COMM SREFP 3 C00296 BC00296  +REFP EC00296
COMM CALL JOB:SEARCH-R1-S13D
COMM SET P032 P006
COMM SFTON3D P032
COMM SMOVL C00297 BC00297 V=166.7  +MOVJ EC00297
COMM SREFP 3 C00298 BC00298  +REFP EC00298
COMM CALL JOB:SEARCH-R1-S13D
COMM SET P032 P006
COMM SFTON3D P032
COMM SMOVL C00299 BC00299 V=166.7  +MOVJ EC00299
COMM SMOVL C00300 BC00300 V=250.0  +MOVJ EC00300
COMM SMOVL C00301 BC00301 V=166.7  +MOVJ EC00301
COMM SREFP 3 C00302 BC00302  +REFP EC00302
COMM CALL JOB:SEARCH-R1-S13D
COMM SET P032 P006
COMM SFTON3D P032
COMM SMOVL C00303 BC00303 V=166.7  +MOVJ EC00303
COMM MOVL C00304 BC00304 V=1000.0  +MOVJ EC00304 VJ=100.00
COMM 'EndPath S4107
COMM '
COMM MOVJ C00305 BC00305 VJ=100.00  +MOVJ EC00305 VJ=100.00
COMM 'Path S4208
COMM SFTOF3D
COMM MOVJ C00306 BC00306 VJ=100.00  +MOVJ EC00306 VJ=100.00
COMM MOVL C00307 BC00307 V=666.7  +MOVJ EC00307 VJ=100.00
COMM SMOVL C00308 BC00308 V=166.7  +MOVJ EC00308
COMM SREFP 3 C00309 BC00309  +REFP EC00309
COMM CALL JOB:SEARCH-R1-S13D
COMM SET P052 P006
COMM SFTON3D P052
COMM SMOVL C00310 BC00310 V=166.7  +MOVJ EC00310
COMM SREFP 3 C00311 BC00311  +REFP EC00311
COMM CALL JOB:SEARCH-R1-S13D
COMM SET P052 P006
COMM SFTON3D P052
COMM SMOVL C00312 BC00312 V=166.7  +MOVJ EC00312
COMM SFTOF3D
COMM MOVL C00313 BC00313 V=1000.0  +MOVJ EC00313 VJ=100.00
COMM SMOVL C00314 BC00314 V=500.0  +MOVJ EC00314
COMM SMOVL C00315 BC00315 V=166.7  +MOVJ EC00315
COMM SREFP 3 C00316 BC00316  +REFP EC00316
COMM CALL JOB:SEARCH-R1-S13D
COMM SET P088 P006
COMM SFTON3D P088
COMM SMOVL C00317 BC00317 V=166.7  +MOVJ EC00317
COMM SMOVL C00318 BC00318 V=166.7  +MOVJ EC00318
COMM SMOVL C00319 BC00319 V=166.7  +MOVJ EC00319
COMM SREFP 3 C00320 BC00320  +REFP EC00320
COMM CALL JOB:SEARCH-R1-S13D
COMM SET P088 P006
COMM SFTON3D P088
COMM SMOVL C00321 BC00321 V=333.3  +MOVJ EC00321
COMM SMOVL C00322 BC00322 V=666.7  +MOVJ EC00322
COMM SFTOF3D
COMM 'EndPath S4208
COMM MOVJ C00323 BC00323 VJ=100.00  +MOVJ EC00323 VJ=100.00
COMM 'Path S4209
COMM SFTOF3D
COMM MOVJ C00324 BC00324 VJ=100.00  +MOVJ EC00324 VJ=100.00
COMM MOVL C00325 BC00325 V=666.7  +MOVJ EC00325 VJ=100.00
COMM SMOVL C00326 BC00326 V=166.7  +MOVJ EC00326
COMM SREFP 3 C00327 BC00327  +REFP EC00327
COMM CALL JOB:SEARCH-R1-S13D
COMM SET P053 P006
COMM SFTON3D P053
COMM SMOVL C00328 BC00328 V=166.7  +MOVJ EC00328
COMM SMOVL C00329 BC00329 V=166.7  +MOVJ EC00329
COMM SREFP 3 C00330 BC00330  +REFP EC00330
COMM CALL JOB:SEARCH-R1-S13D
COMM SET P053 P006
COMM SFTON3D P053
COMM SMOVL C00331 BC00331 V=166.7  +MOVJ EC00331
COMM MOVL C00332 BC00332 V=1000.0  +MOVJ EC00332 VJ=100.00
COMM 'EndPath S4209
COMM *BP1
COMM MOVJ C00333 BC00333 VJ=100.00  +MOVJ EC00333 VJ=100.00
COMM 'Path W4108
COMM SFTOF3D
COMM SFTON3D P033
COMM MOVJ C00334 BC00334 VJ=100.00  +MOVJ EC00334 VJ=100.00
COMM SMOVL C00335 BC00335 V=666.7  +MOVJ EC00335
COMM SMOVL C00336 BC00336 V=166.7 PL=0  +MOVJ EC00336
COMM MACRO1 MJ#(0) ARGF14
COMM ARCON
COMM SMOVL C00337 BC00337 V=9.2  +MOVJ EC00337
COMM ARCOF
COMM SMOVL C00338 BC00338 V=800.0  +MOVJ EC00338
COMM SMOVL C00339 BC00339 V=1000.0  +MOVJ EC00339
COMM SFTOF3D
COMM 'EndPath W4108
COMM 'Path W4109
COMM SFTOF3D
COMM MOVJ C00340 BC00340 VJ=100.00  +MOVJ EC00340 VJ=100.00
COMM MOVJ C00341 BC00341 VJ=100.00  +MOVJ EC00341 VJ=100.00
COMM 'Path W4110
COMM SFTOF3D
COMM SFTON3D P033
COMM MOVJ C00342 BC00342 VJ=100.00  +MOVJ EC00342 VJ=100.00
COMM SMOVL C00343 BC00343 V=800.0  +MOVJ EC00343
COMM SMOVL C00344 BC00344 V=133.3 PL=0  +MOVJ EC00344
COMM MACRO1 MJ#(0) ARGF9
COMM ARCON
COMM SMOVL C00345 BC00345 V=11.7  +MOVJ EC00345
COMM SMOVL C00346 BC00346 V=11.7  +MOVJ EC00346
COMM SMOVL C00347 BC00347 V=11.7  +MOVJ EC00347
COMM ARCOF
COMM SMOVL C00348 BC00348 V=800.0  +MOVJ EC00348
COMM SMOVL C00349 BC00349 V=1000.0  +MOVJ EC00349
COMM SFTOF3D
COMM 'EndPath W4110
COMM MOVJ C00350 BC00350 VJ=100.00  +MOVJ EC00350 VJ=100.00
COMM '9
COMM MOVJ C00351 BC00351 VJ=100.00  +MOVJ EC00351 VJ=100.00
COMM 'Path W4111
COMM SFTOF3D
COMM SFTON3D P026
COMM MOVJ C00352 BC00352 VJ=100.00  +MOVJ EC00352 VJ=100.00
COMM SMOVL C00353 BC00353 V=666.7  +MOVJ EC00353
COMM SMOVL C00354 BC00354 V=166.7 PL=0  +MOVJ EC00354
COMM MACRO1 MJ#(0) ARGF14
COMM ARCON
COMM SMOVL C00355 BC00355 V=9.2  +MOVJ EC00355
COMM ARCOF
COMM SMOVL C00356 BC00356 V=800.0  +MOVJ EC00356
COMM SMOVL C00357 BC00357 V=1000.0  +MOVJ EC00357
COMM SFTOF3D
COMM 'EndPath W4111
COMM 'Path W4112
COMM SFTOF3D
COMM SFTON3D P026
COMM MOVJ C00358 BC00358 VJ=100.00  +MOVJ EC00358 VJ=100.00
COMM SMOVL C00359 BC00359 V=800.0  +MOVJ EC00359
COMM SMOVL C00360 BC00360 V=150.0 PL=0  +MOVJ EC00360
COMM ARCON
COMM SMOVL C00361 BC00361 V=11.7  +MOVJ EC00361
COMM SMOVL C00362 BC00362 V=11.7  +MOVJ EC00362
COMM SMOVL C00363 BC00363 V=11.7  +MOVJ EC00363
COMM ARCOF
COMM SMOVL C00364 BC00364 V=800.0  +MOVJ EC00364
COMM SMOVL C00365 BC00365 V=1000.0  +MOVJ EC00365
COMM SFTOF3D
COMM MOVJ C00366 BC00366 VJ=100.00  +MOVJ EC00366 VJ=100.00
COMM MOVJ C00367 BC00367 VJ=100.00  +MOVJ EC00367 VJ=100.00
COMM 'uwaga na podajnik
COMM 'Path W4114
COMM SFTOF3D
COMM SFTON3D P026
COMM MOVJ C00368 BC00368 VJ=100.00  +MOVJ EC00368 VJ=100.00
COMM SMOVL C00369 BC00369 V=800.0  +MOVJ EC00369
COMM SMOVL C00370 BC00370 V=150.0 PL=0  +MOVJ EC00370
COMM ARCON
COMM SMOVL C00371 BC00371 V=11.7  +MOVJ EC00371
COMM ARCOF
COMM SMOVL C00372 BC00372 V=800.0  +MOVJ EC00372
COMM SMOVL C00373 BC00373 V=1000.0  +MOVJ EC00373
COMM SFTOF3D
COMM 'EndPath W4114
COMM 'brak dostepu offset drutu 1cm
COMM 'Path W4115
COMM SFTOF3D
COMM SFTON3D P026
COMM MOVJ C00374 BC00374 VJ=100.00  +MOVJ EC00374 VJ=100.00
COMM SMOVL C00375 BC00375 V=800.0  +MOVJ EC00375
COMM SMOVL C00376 BC00376 V=150.0 PL=0  +MOVJ EC00376
COMM ARCON
COMM SMOVL C00377 BC00377 V=11.7  +MOVJ EC00377
COMM ARCOF
COMM SMOVL C00378 BC00378 V=800.0  +MOVJ EC00378
COMM SMOVL C00379 BC00379 V=1000.0  +MOVJ EC00379
COMM SFTOF3D
COMM 'EndPath W4115
COMM MOVJ C00380 BC00380 VJ=100.00  +MOVJ EC00380 VJ=100.00
COMM '10
COMM '11
COMM MOVJ C00381 BC00381 VJ=100.00  +MOVJ EC00381 VJ=100.00
COMM 'Path W4118
COMM SFTOF3D
COMM SFTON3D P025
COMM MOVJ C00382 BC00382 VJ=100.00  +MOVJ EC00382 VJ=100.00
COMM SMOVL C00383 BC00383 V=800.0  +MOVJ EC00383
COMM SMOVL C00384 BC00384 V=166.7  +MOVJ EC00384
COMM ARCON
COMM SMOVL C00385 BC00385 V=9.2  +MOVJ EC00385
COMM SMOVL C00386 BC00386 V=9.2  +MOVJ EC00386
COMM SMOVL C00387 BC00387 V=9.2  +MOVJ EC00387
COMM SMOVL C00388 BC00388 V=9.2  +MOVJ EC00388
COMM SMOVL C00389 BC00389 V=9.2  +MOVJ EC00389
COMM ARCOF
COMM SMOVL C00390 BC00390 V=800.0  +MOVJ EC00390
COMM SMOVL C00391 BC00391 V=1000.0  +MOVJ EC00391
COMM SFTOF3D
COMM 'EndPath W4118
COMM 'brak dostepu offset drutu 1cm
COMM MOVJ C00392 BC00392 VJ=100.00  +MOVJ EC00392 VJ=100.00
COMM 'Path W4117
COMM SFTOF3D
COMM SFTON3D P025
COMM MOVJ C00393 BC00393 VJ=100.00  +MOVJ EC00393 VJ=100.00
COMM SMOVL C00394 BC00394 V=800.0  +MOVJ EC00394
COMM SMOVL C00395 BC00395 V=166.7 PL=0  +MOVJ EC00395
COMM ARCON
COMM SMOVL C00396 BC00396 V=10.0  +MOVJ EC00396
COMM ARCOF
COMM SMOVL C00397 BC00397 V=800.0  +MOVJ EC00397
COMM SMOVL C00398 BC00398 V=1000.0  +MOVJ EC00398
COMM SFTOF3D
COMM 'EndPath W4117
COMM '12
COMM MOVJ C00399 BC00399 VJ=100.00  +MOVJ EC00399 VJ=100.00
COMM MOVJ C00400 BC00400 VJ=100.00  +MOVJ EC00400 VJ=100.00
COMM 'Path W4859
COMM SFTOF3D
COMM SFTON3D P073
COMM MOVJ C00401 BC00401 VJ=100.00  +MOVJ EC00401 VJ=100.00
COMM SMOVL C00402 BC00402 V=800.0  +MOVJ EC00402
COMM SMOVL C00403 BC00403 V=150.0 PL=0  +MOVJ EC00403
COMM ARCON
COMM SMOVL C00404 BC00404 V=8.3  +MOVJ EC00404
COMM SFTON3D P074
COMM SMOVL C00405 BC00405 V=9.2  +MOVJ EC00405
COMM SMOVL C00406 BC00406 V=9.2  +MOVJ EC00406
COMM ARCOF
COMM SMOVL C00407 BC00407 V=800.0  +MOVJ EC00407
COMM SMOVL C00408 BC00408 V=1000.0  +MOVJ EC00408
COMM SFTOF3D
COMM 'EndPath W4859
COMM MOVJ C00409 BC00409 VJ=100.00  +MOVJ EC00409 VJ=100.00
COMM MOVJ C00410 BC00410 VJ=100.00  +MOVJ EC00410 VJ=100.00
COMM 'Path W4119
COMM SFTOF3D
COMM SFTON3D P034
COMM MOVJ C00411 BC00411 VJ=100.00  +MOVJ EC00411 VJ=100.00
COMM SMOVL C00412 BC00412 V=800.0  +MOVJ EC00412
COMM SMOVL C00413 BC00413 V=150.0 PL=0  +MOVJ EC00413
COMM ARCON
COMM SMOVL C00414 BC00414 V=10.0  +MOVJ EC00414
COMM SMOVL C00415 BC00415 V=10.0  +MOVJ EC00415
COMM SMOVL C00416 BC00416 V=10.0  +MOVJ EC00416
COMM ARCOF
COMM SMOVL C00417 BC00417 V=800.0  +MOVJ EC00417
COMM SMOVL C00418 BC00418 V=1000.0  +MOVJ EC00418
COMM SFTOF3D
COMM 'EndPath W4119
COMM 'Path W4210
COMM SFTOF3D
COMM SFTON3D P050
COMM MOVJ C00419 BC00419 VJ=100.00  +MOVJ EC00419 VJ=100.00
COMM SMOVL C00420 BC00420 V=800.0  +MOVJ EC00420
COMM SMOVL C00421 BC00421 V=150.0 PL=0  +MOVJ EC00421
COMM ARCON
COMM SMOVL C00422 BC00422 V=11.7  +MOVJ EC00422
COMM ARCOF
COMM SMOVL C00423 BC00423 V=800.0  +MOVJ EC00423
COMM SMOVL C00424 BC00424 V=1000.0  +MOVJ EC00424
COMM SFTOF3D
COMM 'EndPath W4210
COMM 'Path W4211
COMM SFTOF3D
COMM SFTON3D P034
COMM MOVJ C00425 BC00425 VJ=100.00  +MOVJ EC00425 VJ=100.00
COMM SMOVL C00426 BC00426 V=800.0  +MOVJ EC00426
COMM SMOVL C00427 BC00427 V=166.7 PL=0  +MOVJ EC00427
COMM ARCON
COMM SWVON WEV#(66)
COMM SMOVL C00428 BC00428 V=9.2  +MOVJ EC00428
COMM SMOVL C00429 BC00429 V=9.2  +MOVJ EC00429
COMM SMOVL C00430 BC00430 V=9.2  +MOVJ EC00430
COMM ARCOF
COMM SMOVL C00431 BC00431 V=800.0  +MOVJ EC00431
COMM SMOVL C00432 BC00432 V=1000.0  +MOVJ EC00432
COMM MOVJ C00433 BC00433 VJ=30.00  +MOVJ EC00433 VJ=30.00
COMM MOVJ C00434 BC00434 VJ=30.00  +MOVJ EC00434 VJ=30.00
COMM SFTOF3D
COMM MACRO1 MJ#(0) ARGF6
COMM MOVJ C00435 BC00435 VJ=30.00  +MOVJ EC00435 VJ=30.00
COMM SFTON3D P063
COMM SMOVL C00436 BC00436 V=133.3  +MOVJ EC00436
COMM ARCON
COMM SMOVL C00437 BC00437 V=11.7  +MOVJ EC00437
COMM SMOVL C00438 BC00438 V=11.7  +MOVJ EC00438
COMM SMOVL C00439 BC00439 V=11.7  +MOVJ EC00439
COMM SFTON3D P062
COMM SMOVL C00440 BC00440 V=11.7  +MOVJ EC00440
COMM SMOVL C00441 BC00441 V=11.7  +MOVJ EC00441
COMM SFTON3D P061
COMM SMOVL C00442 BC00442 V=11.0  +MOVJ EC00442
COMM SMOVL C00443 BC00443 V=11.0  +MOVJ EC00443
COMM ARCOF
COMM SMOVL C00444 BC00444 V=250.0  +MOVJ EC00444
COMM SFTOF3D
COMM MOVJ C00445 BC00445 VJ=30.00  +MOVJ EC00445 VJ=30.00
COMM MOVJ C00446 BC00446 VJ=30.00  +MOVJ EC00446 VJ=30.00
COMM 'EndPath W4211
COMM 'Path W4210
COMM SFTOF3D
COMM SFTON3D P054
COMM MOVJ C00447 BC00447 VJ=100.00  +MOVJ EC00447 VJ=100.00
COMM SMOVL C00448 BC00448 V=800.0  +MOVJ EC00448
COMM SMOVL C00449 BC00449 V=150.0 PL=0  +MOVJ EC00449
COMM MACRO1 MJ#(0) ARGF14
COMM ARCON
COMM SWVON WEV#(67)
COMM SMOVL C00450 BC00450 V=10.0  +MOVJ EC00450
COMM SMOVL C00451 BC00451 V=10.0  +MOVJ EC00451
COMM ARCOF
COMM SWVOF
COMM SMOVL C00452 BC00452 V=800.0  +MOVJ EC00452
COMM SMOVL C00453 BC00453 V=1000.0  +MOVJ EC00453
COMM SFTOF3D
COMM 'EndPath W4210
COMM 'Path W4121
COMM SFTOF3D
COMM SFTON3D P028
COMM MOVJ C00454 BC00454 VJ=100.00  +MOVJ EC00454 VJ=100.00
COMM SMOVL C00455 BC00455 V=800.0  +MOVJ EC00455
COMM SMOVL C00456 BC00456 V=150.0 PL=0  +MOVJ EC00456
COMM ARCON
COMM SMOVL C00457 BC00457 V=9.2  +MOVJ EC00457
COMM SMOVL C00458 BC00458 V=9.2  +MOVJ EC00458
COMM SMOVL C00459 BC00459 V=9.2  +MOVJ EC00459
COMM ARCOF
COMM SMOVL C00460 BC00460 V=800.0  +MOVJ EC00460
COMM SMOVL C00461 BC00461 V=1000.0  +MOVJ EC00461
COMM SFTOF3D
COMM 'EndPath W4121
COMM 'brak dostepu offset 5mm
COMM MOVJ C00462 BC00462 VJ=100.00  +MOVJ EC00462 VJ=100.00
COMM 'Path W4122
COMM SFTOF3D
COMM SFTON3D P028
COMM MOVJ C00463 BC00463 VJ=100.00  +MOVJ EC00463 VJ=100.00
COMM SMOVL C00464 BC00464 V=800.0  +MOVJ EC00464
COMM SMOVL C00465 BC00465 V=166.7 PL=0  +MOVJ EC00465
COMM ARCON
COMM SMOVL C00466 BC00466 V=11.7  +MOVJ EC00466
COMM ARCOF
COMM SMOVL C00467 BC00467 V=800.0  +MOVJ EC00467
COMM SMOVL C00468 BC00468 V=1000.0  +MOVJ EC00468
COMM SFTOF3D
COMM 'EndPath W4122
COMM MOVJ C00469 BC00469 VJ=100.00  +MOVJ EC00469 VJ=100.00
COMM '13
COMM MOVJ C00470 BC00470 VJ=100.00  +MOVJ EC00470 VJ=100.00
COMM 'Path W4123
COMM SFTOF3D
COMM SFTON3D P030
COMM MOVJ C00471 BC00471 VJ=100.00  +MOVJ EC00471 VJ=100.00
COMM SMOVL C00472 BC00472 V=800.0  +MOVJ EC00472
COMM SMOVL C00473 BC00473 V=150.0 PL=0  +MOVJ EC00473
COMM MACRO1 MJ#(0) ARGF9
COMM ARCON
COMM SWVON WEV#(10)
COMM SFTON3D P031
COMM SMOVL C00474 BC00474 V=12.5  +MOVJ EC00474
COMM ARCOF
COMM SWVOF
COMM SMOVL C00475 BC00475 V=800.0  +MOVJ EC00475
COMM SMOVL C00476 BC00476 V=1000.0  +MOVJ EC00476
COMM SFTOF3D
COMM 'EndPath W4123
COMM '14
COMM '15-brak
COMM 'Path W4212
COMM SFTOF3D
COMM SFTON3D P052
COMM MOVJ C00477 BC00477 VJ=100.00  +MOVJ EC00477 VJ=100.00
COMM SMOVL C00478 BC00478 V=800.0  +MOVJ EC00478
COMM SMOVL C00479 BC00479 V=150.0 PL=0  +MOVJ EC00479
COMM ARCON
COMM SMOVL C00480 BC00480 V=10.8  +MOVJ EC00480
COMM SMOVL C00481 BC00481 V=10.8  +MOVJ EC00481
COMM SMOVL C00482 BC00482 V=10.8  +MOVJ EC00482
COMM ARCOF
COMM SMOVL C00483 BC00483 V=800.0  +MOVJ EC00483
COMM MACRO1 MJ#(0) ARGF6
COMM SMOVL C00484 BC00484 V=333.3  +MOVJ EC00484
COMM SFTOF3D
COMM 'DODAC SHIFT
COMM SFTON3D P088
COMM SMOVL C00485 BC00485 V=133.3  +MOVJ EC00485
COMM ARCON
COMM SMOVL C00486 BC00486 V=10.8  +MOVJ EC00486
COMM ARCOF
COMM SMOVL C00487 BC00487 V=250.0  +MOVJ EC00487
COMM SMOVL C00488 BC00488 V=1000.0  +MOVJ EC00488
COMM SFTOF3D
COMM 'EndPath W4212
COMM '16
COMM 'Path W4213
COMM SFTOF3D
COMM SFTON3D P053
COMM MOVJ C00489 BC00489 VJ=100.00  +MOVJ EC00489 VJ=100.00
COMM SMOVL C00490 BC00490 V=800.0  +MOVJ EC00490
COMM SMOVL C00491 BC00491 V=150.0 PL=0  +MOVJ EC00491
COMM MACRO1 MJ#(0) ARGF9
COMM ARCON
COMM SMOVL C00492 BC00492 V=10.8  +MOVJ EC00492
COMM SMOVL C00493 BC00493 V=10.8  +MOVJ EC00493
COMM SMOVL C00494 BC00494 V=10.8  +MOVJ EC00494
COMM ARCOF
COMM SMOVL C00495 BC00495 V=800.0  +MOVJ EC00495
COMM SMOVL C00496 BC00496 V=1000.0  +MOVJ EC00496
COMM SFTOF3D
COMM 'EndPath W4213
COMM 'Path W4124
COMM SFTOF3D
COMM SFTON3D P029
COMM MOVJ C00497 BC00497 VJ=100.00  +MOVJ EC00497 VJ=100.00
COMM SMOVL C00498 BC00498 V=800.0  +MOVJ EC00498
COMM SMOVL C00499 BC00499 V=166.7 PL=0  +MOVJ EC00499
COMM MACRO1 MJ#(0) ARGF14
COMM ARCON
COMM SMOVL C00500 BC00500 V=10.0  +MOVJ EC00500
COMM SMOVL C00501 BC00501 V=10.0  +MOVJ EC00501
COMM ARCOF
COMM SMOVL C00502 BC00502 V=800.0  +MOVJ EC00502
COMM SMOVL C00503 BC00503 V=1000.0  +MOVJ EC00503
COMM SFTOF3D
COMM 'EndPath W4124
COMM MOVJ C00504 BC00504 VJ=100.00  +MOVJ EC00504 VJ=100.00
COMM 'Path W4125
COMM SFTOF3D
COMM SFTON3D P029
COMM MOVJ C00505 BC00505 VJ=100.00  +MOVJ EC00505 VJ=100.00
COMM SMOVL C00506 BC00506 V=800.0  +MOVJ EC00506
COMM SMOVL C00507 BC00507 V=150.0 PL=0  +MOVJ EC00507
COMM ARCON
COMM SMOVL C00508 BC00508 V=11.7  +MOVJ EC00508
COMM SMOVL C00509 BC00509 V=11.7  +MOVJ EC00509
COMM SMOVL C00510 BC00510 V=11.7  +MOVJ EC00510
COMM ARCOF
COMM SMOVL C00511 BC00511 V=800.0  +MOVJ EC00511
COMM SMOVL C00512 BC00512 V=1000.0  +MOVJ EC00512
COMM SFTOF3D
COMM 'EndPath W4125
COMM MOVJ C00513 BC00513 VJ=100.00  +MOVJ EC00513 VJ=100.00
COMM 'Path W4126
COMM SFTOF3D
COMM SFTON3D P029
COMM MOVJ C00514 BC00514 VJ=100.00  +MOVJ EC00514 VJ=100.00
COMM SMOVL C00515 BC00515 V=800.0  +MOVJ EC00515
COMM SMOVL C00516 BC00516 V=166.7 PL=0  +MOVJ EC00516
COMM ARCON
COMM SMOVL C00517 BC00517 V=11.7  +MOVJ EC00517
COMM ARCON
COMM SMOVL C00518 BC00518 V=11.7  +MOVJ EC00518
COMM SMOVL C00519 BC00519 V=11.7  +MOVJ EC00519
COMM ARCOF
COMM SMOVL C00520 BC00520 V=800.0  +MOVJ EC00520
COMM SMOVL C00521 BC00521 V=1000.0  +MOVJ EC00521
COMM SFTOF3D
COMM 'EndPath W4126
COMM MOVJ C00522 BC00522 VJ=100.00  +MOVJ EC00522 VJ=100.00
COMM '17
COMM 'Path W4127
COMM SFTOF3D
COMM SFTON3D P027
COMM MOVJ C00523 BC00523 VJ=100.00  +MOVJ EC00523 VJ=100.00
COMM SMOVL C00524 BC00524 V=800.0  +MOVJ EC00524
COMM SMOVL C00525 BC00525 V=150.0 PL=0  +MOVJ EC00525
COMM ARCON
COMM SMOVL C00526 BC00526 V=10.0  +MOVJ EC00526
COMM ARCOF
COMM SMOVL C00527 BC00527 V=800.0  +MOVJ EC00527
COMM SMOVL C00528 BC00528 V=1000.0  +MOVJ EC00528
COMM SFTOF3D
COMM 'EndPath W4127
COMM 'Path W4128
COMM SFTOF3D
COMM SFTON3D P027
COMM MOVJ C00529 BC00529 VJ=100.00  +MOVJ EC00529 VJ=100.00
COMM SMOVL C00530 BC00530 V=800.0  +MOVJ EC00530
COMM SMOVL C00531 BC00531 V=150.0 PL=0  +MOVJ EC00531
COMM ARCON
COMM SMOVL C00532 BC00532 V=11.7  +MOVJ EC00532
COMM ARCOF
COMM SMOVL C00533 BC00533 V=800.0  +MOVJ EC00533
COMM SMOVL C00534 BC00534 V=1000.0  +MOVJ EC00534
COMM SFTOF3D
COMM 'EndPath W4128
COMM 'Path W4129
COMM SFTOF3D
COMM SFTON3D P027
COMM MOVJ C00535 BC00535 VJ=100.00  +MOVJ EC00535 VJ=100.00
COMM SMOVL C00536 BC00536 V=800.0  +MOVJ EC00536
COMM SMOVL C00537 BC00537 V=150.0 PL=0  +MOVJ EC00537
COMM SMOVL C00538 BC00538 V=16.7  +MOVJ EC00538
COMM ARCOF
COMM SMOVL C00539 BC00539 V=800.0  +MOVJ EC00539
COMM SMOVL C00540 BC00540 V=1000.0  +MOVJ EC00540
COMM SFTOF3D
COMM 'EndPath W4129
COMM '18
COMM MOVJ C00541 BC00541 VJ=100.00  +MOVJ EC00541 VJ=100.00
COMM 'Path W4130
COMM SFTOF3D
COMM SFTON3D P024
COMM MOVJ C00542 BC00542 VJ=100.00  +MOVJ EC00542 VJ=100.00
COMM SMOVL C00543 BC00543 V=800.0  +MOVJ EC00543
COMM SMOVL C00544 BC00544 V=150.0 PL=0  +MOVJ EC00544
COMM ARCON
COMM SMOVL C00545 BC00545 V=9.2  +MOVJ EC00545
COMM SMOVL C00546 BC00546 V=9.2  +MOVJ EC00546
COMM SMOVL C00547 BC00547 V=9.2  +MOVJ EC00547
COMM SMOVL C00548 BC00548 V=9.2  +MOVJ EC00548
COMM ARCOF
COMM SMOVL C00549 BC00549 V=800.0  +MOVJ EC00549
COMM SMOVL C00550 BC00550 V=1000.0  +MOVJ EC00550
COMM SFTOF3D
COMM 'EndPath W4130
COMM 'Path W4860
COMM SFTOF3D
COMM SFTON3D P071
COMM MOVJ C00551 BC00551 VJ=100.00  +MOVJ EC00551 VJ=100.00
COMM SMOVL C00552 BC00552 V=800.0  +MOVJ EC00552
COMM SMOVL C00553 BC00553 V=150.0 PL=0  +MOVJ EC00553
COMM MACRO1 MJ#(0) ARGF9
COMM ARCON
COMM SMOVL C00554 BC00554 V=9.2  +MOVJ EC00554
COMM SFTON3D P072
COMM ARCON
COMM SMOVL C00555 BC00555 V=9.2  +MOVJ EC00555
COMM SMOVL C00556 BC00556 V=9.2  +MOVJ EC00556
COMM ARCOF
COMM SMOVL C00557 BC00557 V=800.0  +MOVJ EC00557
COMM SMOVL C00558 BC00558 V=1000.0  +MOVJ EC00558
COMM SFTOF3D
COMM 'EndPath W4860
COMM '19
COMM MOVJ C00559 BC00559 VJ=100.00  +MOVJ EC00559 VJ=100.00
COMM 'Path W4131
COMM SFTOF3D
COMM SFTON3D P023
COMM MOVJ C00560 BC00560 VJ=100.00  +MOVJ EC00560 VJ=100.00
COMM SMOVL C00561 BC00561 V=800.0  +MOVJ EC00561
COMM SMOVL C00562 BC00562 V=166.7 PL=0  +MOVJ EC00562
COMM MACRO1 MJ#(0) ARGF9
COMM ARCON
COMM SWVON WEV#(60)
COMM SMOVL C00563 BC00563 V=7.5  +MOVJ EC00563
COMM SMOVL C00564 BC00564 V=7.5  +MOVJ EC00564
COMM SMOVL C00565 BC00565 V=7.5  +MOVJ EC00565
COMM ARCOF
COMM SWVOF
COMM SMOVL C00566 BC00566 V=800.0  +MOVJ EC00566
COMM SMOVL C00567 BC00567 V=1000.0  +MOVJ EC00567
COMM SFTOF3D
COMM 'EndPath W4131
COMM MOVJ C00568 BC00568 VJ=100.00  +MOVJ EC00568 VJ=100.00
COMM 'Path W4214
COMM SFTOF3D
COMM SFTON3D P089
COMM MOVJ C00569 BC00569 VJ=100.00  +MOVJ EC00569 VJ=100.00
COMM SMOVL C00570 BC00570 V=800.0  +MOVJ EC00570
COMM SMOVL C00571 BC00571 V=150.0 PL=0  +MOVJ EC00571
COMM MACRO1 MJ#(0) ARGF9
COMM ARCON
COMM SMOVL C00572 BC00572 V=9.2  +MOVJ EC00572
COMM SFTON3D P050
COMM SMOVL C00573 BC00573 V=9.2  +MOVJ EC00573
COMM SMOVL C00574 BC00574 V=9.2  +MOVJ EC00574
COMM ARCOF
COMM SMOVL C00575 BC00575 V=800.0  +MOVJ EC00575
COMM SMOVL C00576 BC00576 V=1000.0  +MOVJ EC00576
COMM SFTOF3D
COMM 'EndPath W4214
COMM 'Path W4215
COMM SFTOF3D
COMM SFTON3D P051
COMM MOVJ C00577 BC00577 VJ=100.00  +MOVJ EC00577 VJ=100.00
COMM SMOVL C00578 BC00578 V=800.0  +MOVJ EC00578
COMM SMOVL C00579 BC00579 V=150.0 PL=0  +MOVJ EC00579
COMM MACRO1 MJ#(0) ARGF9
COMM ARCON
COMM SWVON WEV#(60)
COMM SMOVL C00580 BC00580 V=7.5  +MOVJ EC00580
COMM SMOVL C00581 BC00581 V=7.5  +MOVJ EC00581
COMM SMOVL C00582 BC00582 V=7.5  +MOVJ EC00582
COMM ARCOF
COMM SWVOF
COMM SMOVL C00583 BC00583 V=800.0  +MOVJ EC00583
COMM SMOVL C00584 BC00584 V=1000.0  +MOVJ EC00584
COMM SFTOF3D
COMM 'EndPath W4215
COMM MOVJ C00585 BC00585 VJ=100.00  +MOVJ EC00585 VJ=100.00
COMM '20
COMM 'offset 5mm
COMM MOVJ C00586 BC00586 VJ=100.00  +MOVJ EC00586 VJ=100.00
COMM MOVJ C00587 BC00587 VJ=100.00  +MOVJ EC00587 VJ=100.00
COMM 'Path W4132
COMM SFTOF3D
COMM SFTON3D P032
COMM MOVJ C00588 BC00588 VJ=100.00  +MOVJ EC00588 VJ=100.00
COMM SMOVL C00589 BC00589 V=800.0  +MOVJ EC00589
COMM SMOVL C00590 BC00590 V=150.0 PL=0  +MOVJ EC00590
COMM ARCON
COMM SMOVL C00591 BC00591 V=10.0  +MOVJ EC00591
COMM SMOVL C00592 BC00592 V=10.0  +MOVJ EC00592
COMM ARCOF
COMM SMOVL C00593 BC00593 V=800.0  +MOVJ EC00593
COMM SMOVL C00594 BC00594 V=1000.0  +MOVJ EC00594
COMM SFTOF3D
COMM JUMP *FFF
COMM 'EndPath W4132
COMM 'Path W4133
COMM SFTOF3D
COMM SFTON3D P032
COMM MOVJ C00595 BC00595 VJ=100.00  +MOVJ EC00595 VJ=100.00
COMM SMOVL C00596 BC00596 V=800.0  +MOVJ EC00596
COMM SMOVL C00597 BC00597 V=166.7 PL=0  +MOVJ EC00597
COMM ARCON
COMM SMOVL C00598 BC00598 V=10.0  +MOVJ EC00598
COMM ARCOF
COMM SMOVL C00599 BC00599 V=800.0  +MOVJ EC00599
COMM SMOVL C00600 BC00600 V=1000.0  +MOVJ EC00600
COMM SFTOF3D
COMM 'EndPath W4133
COMM 'Path W4134
COMM SFTOF3D
COMM SFTON3D P032
COMM MOVJ C00601 BC00601 VJ=100.00  +MOVJ EC00601 VJ=100.00
COMM SMOVL C00602 BC00602 V=800.0  +MOVJ EC00602
COMM SMOVL C00603 BC00603 V=150.0 PL=0  +MOVJ EC00603
COMM ARCON
COMM SMOVL C00604 BC00604 V=10.0  +MOVJ EC00604
COMM ARCOF
COMM SMOVL C00605 BC00605 V=800.0  +MOVJ EC00605
COMM *FFF
COMM SMOVL C00606 BC00606 V=1000.0  +MOVJ EC00606
COMM SFTOF3D
COMM 'EndPath W4134
COMM 'offset 5mm
COMM MOVJ C00607 BC00607 VJ=100.00  +MOVJ EC00607 VJ=100.00
COMM 'Path W4135
COMM SFTOF3D
COMM SFTON3D P032
COMM MOVJ C00608 BC00608 VJ=100.00  +MOVJ EC00608 VJ=100.00
COMM SMOVL C00609 BC00609 V=800.0  +MOVJ EC00609
COMM SMOVL C00610 BC00610 V=166.7 PL=0  +MOVJ EC00610
COMM ARCON
COMM SMOVL C00611 BC00611 V=10.0  +MOVJ EC00611
COMM ARCOF
COMM SMOVL C00612 BC00612 V=800.0  +MOVJ EC00612
COMM SMOVL C00613 BC00613 V=1000.0  +MOVJ EC00613
COMM SFTOF3D
COMM 'EndPath W4135
COMM MOVJ C00614 BC00614 VJ=100.00  +MOVJ EC00614 VJ=100.00
COMM 'Path W4136
COMM SFTOF3D
COMM SFTON3D P032
COMM MOVJ C00615 BC00615 VJ=100.00  +MOVJ EC00615 VJ=100.00
COMM SMOVL C00616 BC00616 V=800.0  +MOVJ EC00616
COMM SMOVL C00617 BC00617 V=166.7 PL=0  +MOVJ EC00617
COMM ARCON
COMM SMOVL C00618 BC00618 V=11.7  +MOVJ EC00618
COMM SMOVL C00619 BC00619 V=11.7  +MOVJ EC00619
COMM ARCOF
COMM SMOVL C00620 BC00620 V=800.0  +MOVJ EC00620
COMM SMOVL C00621 BC00621 V=1000.0  +MOVJ EC00621
COMM SFTOF3D
COMM 'EndPath W4136
COMM MOVJ C00622 BC00622 VJ=100.00  +MOVJ EC00622 VJ=100.00
COMM MOVJ C00623 BC00623 VJ=100.00  +MOVJ EC00623 VJ=100.00
COMM 'Path W4137
COMM SFTOF3D
COMM SFTON3D P021
COMM MOVJ C00624 BC00624 VJ=100.00  +MOVJ EC00624 VJ=100.00
COMM SMOVL C00625 BC00625 V=800.0  +MOVJ EC00625
COMM SMOVL C00626 BC00626 V=150.0 PL=0  +MOVJ EC00626
COMM MACRO1 MJ#(0) ARGF9
COMM ARCON
COMM SFTON3D P022
COMM SMOVL C00627 BC00627 V=10.0  +MOVJ EC00627
COMM ARCOF
COMM SMOVL C00628 BC00628 V=800.0  +MOVJ EC00628
COMM SMOVL C00629 BC00629 V=1000.0  +MOVJ EC00629
COMM SFTOF3D
COMM 'EndPath W4137
COMM MOVJ C00630 BC00630 VJ=100.00  +MOVJ EC00630 VJ=100.00
COMM 'Path W4724
COMM SFTOF3D
COMM SFTON3D P095
COMM MOVJ C00631 BC00631 VJ=100.00  +MOVJ EC00631 VJ=100.00
COMM SMOVL C00632 BC00632 V=800.0  +MOVJ EC00632
COMM SMOVL C00633 BC00633 V=150.0 PL=0  +MOVJ EC00633
COMM ARCON
COMM SMOVL C00634 BC00634 V=10.0  +MOVJ EC00634
COMM SMOVL C00635 BC00635 V=10.0  +MOVJ EC00635
COMM SMOVL C00636 BC00636 V=10.0  +MOVJ EC00636
COMM ARCOF
COMM SMOVL C00637 BC00637 V=800.0  +MOVJ EC00637
COMM SMOVL C00638 BC00638 V=1000.0  +MOVJ EC00638
COMM SFTOF3D
COMM 'EndPath W4724
COMM 'Path W4725
COMM SFTOF3D
COMM SFTON3D P096
COMM MOVJ C00639 BC00639 VJ=100.00  +MOVJ EC00639 VJ=100.00
COMM SMOVL C00640 BC00640 V=800.0  +MOVJ EC00640
COMM SMOVL C00641 BC00641 V=150.0 PL=0  +MOVJ EC00641
COMM ARCON
COMM SMOVL C00642 BC00642 V=10.0  +MOVJ EC00642
COMM SMOVL C00643 BC00643 V=10.0  +MOVJ EC00643
COMM ARCOF
COMM SMOVL C00644 BC00644 V=800.0  +MOVJ EC00644
COMM SMOVL C00645 BC00645 V=1000.0  +MOVJ EC00645
COMM SFTOF3D
COMM 'EndPath W4725
COMM MOVJ C00646 BC00646 VJ=100.00  +MOVJ EC00646 VJ=100.00
COMM 'Path W4861
COMM SFTOF3D
COMM SFTON3D P071
COMM MOVJ C00647 BC00647 VJ=100.00  +MOVJ EC00647 VJ=100.00
COMM SMOVL C00648 BC00648 V=800.0  +MOVJ EC00648
COMM SMOVL C00649 BC00649 V=150.0 PL=0  +MOVJ EC00649
COMM MACRO1 MJ#(0) ARGF14
COMM ARCON
COMM SMOVL C00650 BC00650 V=9.2  +MOVJ EC00650
COMM SFTON3D P073
COMM SMOVL C00651 BC00651 V=9.2  +MOVJ EC00651
COMM SMOVL C00652 BC00652 V=9.2  +MOVJ EC00652
COMM ARCOF
COMM SMOVL C00653 BC00653 V=800.0  +MOVJ EC00653
COMM SMOVL C00654 BC00654 V=1000.0  +MOVJ EC00654
COMM SFTOF3D
COMM 'EndPath W4861
COMM MOVJ C00655 BC00655 VJ=100.00  +MOVJ EC00655 VJ=100.00
COMM MOVJ C00656 BC00656 VJ=100.00  +MOVJ EC00656 VJ=100.00
'X2_8B-21B(90,180)
'
MOVJ C00657 BC00657 VJ=100.00  +MOVJ EC00657 VJ=100.00
'Path S4722
SFTOF3D
MOVJ C00658 BC00658 VJ=100.00  +MOVJ EC00658 VJ=100.00
MOVL C00659 BC00659 V=666.7  +MOVJ EC00659 VJ=100.00
SMOVL C00660 BC00660 V=166.7  +MOVJ EC00660
SREFP 3 C00661 BC00661  +REFP EC00661
CALL JOB:SEARCH-R1-S13D
SET P095 P006
SFTON3D P095
SMOVL C00662 BC00662 V=166.7  +MOVJ EC00662
SREFP 3 C00663 BC00663  +REFP EC00663
CALL JOB:SEARCH-R1-S13D
SET P095 P006
SFTON3D P095
SMOVL C00664 BC00664 V=166.7  +MOVJ EC00664
MOVL C00665 BC00665 V=1000.0  +MOVJ EC00665 VJ=100.00
'EndPath S4722
'Path S4723
SFTOF3D
MOVJ C00666 BC00666 VJ=100.00  +MOVJ EC00666 VJ=100.00
MOVL C00667 BC00667 V=666.7  +MOVJ EC00667 VJ=100.00
SMOVL C00668 BC00668 V=166.7  +MOVJ EC00668
SREFP 3 C00669 BC00669  +REFP EC00669
CALL JOB:SEARCH-R1-S13D
SET P096 P006
SFTON3D P096
SMOVL C00670 BC00670 V=166.7  +MOVJ EC00670
SREFP 3 C00671 BC00671  +REFP EC00671
CALL JOB:SEARCH-R1-S13D
SET P096 P006
SFTON3D P096
SMOVL C00672 BC00672 V=166.7  +MOVJ EC00672
MOVL C00673 BC00673 V=1000.0  +MOVJ EC00673 VJ=100.00
'EndPath S4723
'
'
'Path S4093
SFTOF3D
MOVJ C00674 BC00674 VJ=100.00  +MOVJ EC00674 VJ=100.00
MOVL C00675 BC00675 V=666.7  +MOVJ EC00675 VJ=100.00
SMOVL C00676 BC00676 V=166.7  +MOVJ EC00676
SREFP 3 C00677 BC00677  +REFP EC00677
CALL JOB:SEARCH-R1-S13D
SET P097 P006
SFTON3D P097
SMOVL C00678 BC00678 V=166.7  +MOVJ EC00678
SREFP 3 C00679 BC00679  +REFP EC00679
CALL JOB:SEARCH-R1-S13D
SET P097 P006
SFTON3D P097
SMOVL C00680 BC00680 V=166.7  +MOVJ EC00680
SFTOF3D
MOVL C00681 BC00681 V=666.7  +MOVJ EC00681 VJ=100.00
SMOVL C00682 BC00682 V=166.7  +MOVJ EC00682
SREFP 3 C00683 BC00683  +REFP EC00683
CALL JOB:SEARCH-R1-S13D
SET P021 P006
SFTON3D P021
SMOVL C00684 BC00684 V=166.7  +MOVJ EC00684
SREFP 3 C00685 BC00685  +REFP EC00685
CALL JOB:SEARCH-R1-S13D
SET P021 P006
SFTON3D P021
SMOVL C00686 BC00686 V=166.7  +MOVJ EC00686
MOVL C00687 BC00687 V=1000.0  +MOVJ EC00687 VJ=100.00
'EndPath S4093
'Path S4094
SFTOF3D
MOVJ C00688 BC00688 VJ=100.00  +MOVJ EC00688 VJ=100.00
MOVL C00689 BC00689 V=666.7  +MOVJ EC00689 VJ=100.00
SMOVL C00690 BC00690 V=166.7  +MOVJ EC00690
SREFP 3 C00691 BC00691  +REFP EC00691
CALL JOB:SEARCH-R1-S13D
SET P022 P006
SFTON3D P022
SMOVL C00692 BC00692 V=166.7  +MOVJ EC00692
SREFP 3 C00693 BC00693  +REFP EC00693
CALL JOB:SEARCH-R1-S13D
SET P022 P006
SFTON3D P022
SMOVL C00694 BC00694 V=166.7  +MOVJ EC00694
MOVL C00695 BC00695 V=1000.0  +MOVJ EC00695 VJ=100.00
'EndPath S4094
MOVJ C00696 BC00696 VJ=100.00  +MOVJ EC00696 VJ=100.00
'Path S4205
SFTOF3D
MOVJ C00697 BC00697 VJ=100.00  +MOVJ EC00697 VJ=100.00
MOVL C00698 BC00698 V=666.7  +MOVJ EC00698 VJ=100.00
SMOVL C00699 BC00699 V=166.7  +MOVJ EC00699
SREFP 3 C00700 BC00700  +REFP EC00700
CALL JOB:SEARCH-R1-S13D
SET P050 P006
SFTON3D P050
SMOVL C00701 BC00701 V=166.7  +MOVJ EC00701
SREFP 3 C00702 BC00702  +REFP EC00702
CALL JOB:SEARCH-R1-S13D
SET P050 P006
SFTON3D P050
SMOVL C00703 BC00703 V=166.7  +MOVJ EC00703
SMOVL C00704 BC00704 V=250.0  +MOVJ EC00704
SMOVL C00705 BC00705 V=166.7  +MOVJ EC00705
SREFP 3 C00706 BC00706  +REFP EC00706
CALL JOB:SEARCH-R1-S13D
SET P050 P006
SFTON3D P050
SMOVL C00707 BC00707 V=250.0  +MOVJ EC00707
'EndPath S4205
'Path S4206
SFTOF3D
MOVL C00708 BC00708 V=1000.0  +MOVJ EC00708 VJ=100.00
SMOVL C00709 BC00709 V=166.7  +MOVJ EC00709
SREFP 3 C00710 BC00710  +REFP EC00710
CALL JOB:SEARCH-R1-S13D
SET P051 P006
SFTON3D P051
SMOVL C00711 BC00711 V=166.7  +MOVJ EC00711
SREFP 3 C00712 BC00712  +REFP EC00712
CALL JOB:SEARCH-R1-S13D
SET P051 P006
SFTON3D P051
SMOVL C00713 BC00713 V=166.7  +MOVJ EC00713
SMOVL C00714 BC00714 V=250.0  +MOVJ EC00714
SREFP 3 C00715 BC00715  +REFP EC00715
CALL JOB:SEARCH-R1-S13D
SET P051 P006
SFTON3D P051
SMOVL C00716 BC00716 V=250.0  +MOVJ EC00716
MOVL C00717 BC00717 V=1000.0  +MOVJ EC00717 VJ=100.00
'EndPath S4206
MOVJ C00718 BC00718 VJ=100.00  +MOVJ EC00718 VJ=100.00
'Path S4207
SFTOF3D
MOVJ C00719 BC00719 VJ=100.00  +MOVJ EC00719 VJ=100.00
MOVL C00720 BC00720 V=666.7  +MOVJ EC00720 VJ=100.00
SMOVL C00721 BC00721 V=166.7  +MOVJ EC00721
SREFP 3 C00722 BC00722  +REFP EC00722
CALL JOB:SEARCH-R1-S13D
SET P054 P006
SFTON3D P054
SMOVL C00723 BC00723 V=250.0  +MOVJ EC00723
SMOVL C00724 BC00724 V=233.3  +MOVJ EC00724
SMOVL C00725 BC00725 V=166.7  +MOVJ EC00725
SREFP 3 C00726 BC00726  +REFP EC00726
CALL JOB:SEARCH-R1-S13D
SET P054 P006
SFTON3D P054
SMOVL C00727 BC00727 V=166.7  +MOVJ EC00727
SMOVL C00728 BC00728 V=416.7  +MOVJ EC00728
SMOVL C00729 BC00729 V=250.0  +MOVJ EC00729
SREFP 3 C00730 BC00730  +REFP EC00730
CALL JOB:SEARCH-R1-S13D
SET P054 P006
SFTON3D P054
SMOVL C00731 BC00731 V=250.0  +MOVJ EC00731
MOVL C00732 BC00732 V=1000.0  +MOVJ EC00732 VJ=100.00
'EndPath S4207
'Path S4095
SFTOF3D
MOVJ C00733 BC00733 VJ=100.00  +MOVJ EC00733 VJ=100.00
MOVJ C00734 BC00734 VJ=100.00  +MOVJ EC00734 VJ=100.00
SMOVL C00735 BC00735 V=200.0  +MOVJ EC00735
SREFP 3 C00736 BC00736  +REFP EC00736
CALL JOB:SEARCH-R1-S13D
SET P089 P006
SFTON3D P089
SMOVL C00737 BC00737 V=166.7  +MOVJ EC00737
SMOVL C00738 BC00738 V=166.7  +MOVJ EC00738
SREFP 3 C00739 BC00739  +REFP EC00739
CALL JOB:SEARCH-R1-S13D
SET P089 P006
SFTON3D P089
SMOVL C00740 BC00740 V=166.7  +MOVJ EC00740
SMOVL C00741 BC00741 V=166.7  +MOVJ EC00741
SREFP 3 C00742 BC00742  +REFP EC00742
CALL JOB:SEARCH-R1-S13D
SET P089 P006
SFTON3D P089
SMOVL C00743 BC00743 V=166.7  +MOVJ EC00743
SMOVL C00744 BC00744 V=1000.0  +MOVJ EC00744
SFTOF3D
MOVJ C00745 BC00745 VJ=100.00  +MOVJ EC00745 VJ=100.00
MOVL C00746 BC00746 V=666.7  +MOVJ EC00746 VJ=100.00
SMOVL C00747 BC00747 V=166.7  +MOVJ EC00747
SREFP 3 C00748 BC00748  +REFP EC00748
CALL JOB:SEARCH-R1-S13D
SET P034 P006
SFTON3D P034
SMOVL C00749 BC00749 V=250.0  +MOVJ EC00749
SMOVL C00750 BC00750 V=233.3  +MOVJ EC00750
SMOVL C00751 BC00751 V=166.7  +MOVJ EC00751
SREFP 3 C00752 BC00752  +REFP EC00752
CALL JOB:SEARCH-R1-S13D
SET P034 P006
SFTON3D P034
SMOVL C00753 BC00753 V=166.7  +MOVJ EC00753
SMOVL C00754 BC00754 V=166.7  +MOVJ EC00754
SREFP 3 C00755 BC00755  +REFP EC00755
CALL JOB:SEARCH-R1-S13D
SET P034 P006
SFTON3D P034
SMOVL C00756 BC00756 V=166.7  +MOVJ EC00756
MOVJ C00757 BC00757 VJ=50.00  +MOVJ EC00757 VJ=30.00
'EndPath S4095
'Path S4096
SFTOF3D
MOVJ C00758 BC00758 VJ=50.00  +MOVJ EC00758 VJ=30.00
MOVJ C00759 BC00759 VJ=50.00  +MOVJ EC00759 VJ=30.00
MOVJ C00760 BC00760 VJ=50.00  +MOVJ EC00760 VJ=30.00
SMOVL C00761 BC00761 V=166.7  +MOVJ EC00761
SREFP 3 C00762 BC00762  +REFP EC00762
CALL JOB:SEARCH-R1-S13D
SET P061 P006
SFTON3D P061
SMOVL C00763 BC00763 V=166.7  +MOVJ EC00763
SREFP 3 C00764 BC00764  +REFP EC00764
CALL JOB:SEARCH-R1-S13D
SET P061 P006
SFTON3D P061
SMOVL C00765 BC00765 V=166.7  +MOVJ EC00765
SFTOF3D
SMOVL C00766 BC00766 V=666.7  +MOVJ EC00766
SMOVL C00767 BC00767 V=166.7  +MOVJ EC00767
SREFP 3 C00768 BC00768  +REFP EC00768
CALL JOB:SEARCH-R1-S13D
SET P062 P006
SFTON3D P062
SMOVL C00769 BC00769 V=166.7  +MOVJ EC00769
SREFP 3 C00770 BC00770  +REFP EC00770
CALL JOB:SEARCH-R1-S13D
SET P062 P006
SFTON3D P062
SMOVL C00771 BC00771 V=250.0  +MOVJ EC00771
SFTOF3D
SMOVL C00772 BC00772 V=500.0  +MOVJ EC00772
SMOVL C00773 BC00773 V=166.7  +MOVJ EC00773
SREFP 3 C00774 BC00774  +REFP EC00774
CALL JOB:SEARCH-R1-S13D
SET P063 P006
SFTON3D P063
SMOVL C00775 BC00775 V=166.7  +MOVJ EC00775
SREFP 3 C00776 BC00776  +REFP EC00776
CALL JOB:SEARCH-R1-S13D
SET P063 P006
SFTON3D P063
SMOVL C00777 BC00777 V=166.7  +MOVJ EC00777
SFTOF3D
SMOVL C00778 BC00778 V=1000.0  +MOVJ EC00778
MOVJ C00779 BC00779 VJ=100.00  +MOVJ EC00779 VJ=30.00
MOVJ C00780 BC00780 VJ=50.00  +MOVJ EC00780 VJ=30.00
MOVJ C00781 BC00781 VJ=100.00  +MOVJ EC00781 VJ=100.00
MOVL C00782 BC00782 V=666.7  +MOVJ EC00782 VJ=100.00
SMOVL C00783 BC00783 V=166.7  +MOVJ EC00783
SREFP 3 C00784 BC00784  +REFP EC00784
CALL JOB:SEARCH-R1-S13D
SET P023 P006
SFTON3D P023
SMOVL C00785 BC00785 V=166.7  +MOVJ EC00785
SMOVL C00786 BC00786 V=333.3  +MOVJ EC00786
SMOVL C00787 BC00787 V=166.7  +MOVJ EC00787
SREFP 3 C00788 BC00788  +REFP EC00788
CALL JOB:SEARCH-R1-S13D
SET P023 P006
SFTON3D P023
SMOVL C00789 BC00789 V=166.7  +MOVJ EC00789
SMOVL C00790 BC00790 V=166.7  +MOVJ EC00790
SREFP 3 C00791 BC00791  +REFP EC00791
CALL JOB:SEARCH-R1-S13D
SET P023 P006
SFTON3D P023
SMOVL C00792 BC00792 V=166.7  +MOVJ EC00792
MOVL C00793 BC00793 V=1000.0  +MOVJ EC00793 VJ=100.00
'EndPath S4096
MOVJ C00794 BC00794 VJ=100.00  +MOVJ EC00794 VJ=100.00
'Path S4097
SFTOF3D
MOVJ C00795 BC00795 VJ=100.00  +MOVJ EC00795 VJ=100.00
MOVL C00796 BC00796 V=666.7  +MOVJ EC00796 VJ=100.00
SMOVL C00797 BC00797 V=166.7  +MOVJ EC00797
SREFP 3 C00798 BC00798  +REFP EC00798
CALL JOB:SEARCH-R1-S13D
SET P024 P006
SFTON3D P024
SMOVL C00799 BC00799 V=166.7  +MOVJ EC00799
SREFP 3 C00800 BC00800  +REFP EC00800
CALL JOB:SEARCH-R1-S13D
SET P024 P006
SFTON3D P024
SMOVL C00801 BC00801 V=166.7  +MOVJ EC00801
SMOVL C00802 BC00802 V=166.7  +MOVJ EC00802
SREFP 3 C00803 BC00803  +REFP EC00803
CALL JOB:SEARCH-R1-S13D
SET P024 P006
SFTON3D P024
SMOVL C00804 BC00804 V=166.7  +MOVJ EC00804
MOVL C00805 BC00805 V=1000.0  +MOVJ EC00805 VJ=100.00
'EndPath S4097
'Path S4098
SFTOF3D
MOVJ C00806 BC00806 VJ=100.00  +MOVJ EC00806 VJ=100.00
MOVL C00807 BC00807 V=666.7  +MOVJ EC00807 VJ=100.00
SMOVL C00808 BC00808 V=166.7  +MOVJ EC00808
SREFP 3 C00809 BC00809  +REFP EC00809
CALL JOB:SEARCH-R1-S13D
SET P035 P006
SFTON3D P035
SMOVL C00810 BC00810 V=166.7  +MOVJ EC00810
SREFP 3 C00811 BC00811  +REFP EC00811
CALL JOB:SEARCH-R1-S13D
SET P035 P006
SFTON3D P035
SMOVL C00812 BC00812 V=166.7  +MOVJ EC00812
SMOVL C00813 BC00813 V=166.7  +MOVJ EC00813
SMOVL C00814 BC00814 V=166.7  +MOVJ EC00814
SREFP 3 C00815 BC00815  +REFP EC00815
CALL JOB:SEARCH-R1-S13D
SET P035 P006
SFTON3D P035
SMOVL C00816 BC00816 V=166.7  +MOVJ EC00816
MOVL C00817 BC00817 V=1000.0  +MOVJ EC00817 VJ=100.00
'EndPath S4098
'Path S4099
SFTOF3D
MOVJ C00818 BC00818 VJ=100.00  +MOVJ EC00818 VJ=100.00
MOVL C00819 BC00819 V=666.7  +MOVJ EC00819 VJ=100.00
SMOVL C00820 BC00820 V=166.7  +MOVJ EC00820
SREFP 3 C00821 BC00821  +REFP EC00821
CALL JOB:SEARCH-R1-S13D
SET P029 P006
SFTON3D P029
SMOVL C00822 BC00822 V=166.7  +MOVJ EC00822
SREFP 3 C00823 BC00823  +REFP EC00823
CALL JOB:SEARCH-R1-S13D
SET P029 P006
SFTON3D P029
SMOVL C00824 BC00824 V=166.7  +MOVJ EC00824
SMOVL C00825 BC00825 V=250.0  +MOVJ EC00825
SMOVL C00826 BC00826 V=166.7  +MOVJ EC00826
SREFP 3 C00827 BC00827  +REFP EC00827
CALL JOB:SEARCH-R1-S13D
SET P029 P006
SFTON3D P029
SMOVL C00828 BC00828 V=166.7  +MOVJ EC00828
'EndPath S4099
'Path S4855
SFTOF3D
MOVL C00829 BC00829 V=666.7  +MOVJ EC00829 VJ=100.00
SMOVL C00830 BC00830 V=166.7  +MOVJ EC00830
SREFP 3 C00831 BC00831  +REFP EC00831
CALL JOB:SEARCH-R1-S13D
SET P071 P006
SFTON3D P071
SMOVL C00832 BC00832 V=166.7  +MOVJ EC00832
SREFP 3 C00833 BC00833  +REFP EC00833
CALL JOB:SEARCH-R1-S13D
SET P071 P006
SFTON3D P071
SMOVL C00834 BC00834 V=166.7  +MOVJ EC00834
SMOVL C00835 BC00835 V=166.7  +MOVJ EC00835
SREFP 3 C00836 BC00836  +REFP EC00836
CALL JOB:SEARCH-R1-S13D
SET P071 P006
SFTON3D P071
SMOVL C00837 BC00837 V=166.7  +MOVJ EC00837
MOVL C00838 BC00838 V=1000.0  +MOVJ EC00838 VJ=100.00
MOVL C00839 BC00839 V=666.7  +MOVJ EC00839 VJ=100.00
SMOVL C00840 BC00840 V=166.7  +MOVJ EC00840
SREFP 3 C00841 BC00841  +REFP EC00841
CALL JOB:SEARCH-R1-S13D
SET P080 P006
SFTON3D P080
SMOVL C00842 BC00842 V=166.7  +MOVJ EC00842
SREFP 3 C00843 BC00843  +REFP EC00843
CALL JOB:SEARCH-R1-S13D
SET P080 P006
SFTON3D P080
SMOVL C00844 BC00844 V=166.7  +MOVJ EC00844
SMOVL C00845 BC00845 V=250.0  +MOVJ EC00845
SMOVL C00846 BC00846 V=166.7  +MOVJ EC00846
SREFP 3 C00847 BC00847  +REFP EC00847
CALL JOB:SEARCH-R1-S13D
SET P080 P006
SFTON3D P080
SMOVL C00848 BC00848 V=166.7  +MOVJ EC00848
'EndPath S4855
'Path S4856
SFTOF3D
MOVJ C00849 BC00849 VJ=100.00  +MOVJ EC00849 VJ=100.00
MOVL C00850 BC00850 V=666.7  +MOVJ EC00850 VJ=100.00
SMOVL C00851 BC00851 V=166.7  +MOVJ EC00851
SREFP 3 C00852 BC00852  +REFP EC00852
CALL JOB:SEARCH-R1-S13D
SET P072 P006
SFTON3D P072
SMOVL C00853 BC00853 V=166.7  +MOVJ EC00853
SREFP 3 C00854 BC00854  +REFP EC00854
CALL JOB:SEARCH-R1-S13D
SET P072 P006
SFTON3D P072
SMOVL C00855 BC00855 V=166.7  +MOVJ EC00855
MOVL C00856 BC00856 V=1000.0  +MOVJ EC00856 VJ=100.00
'EndPath S4856
MOVJ C00857 BC00857 VJ=100.00  +MOVJ EC00857 VJ=100.00
'Path S4857
SFTOF3D
MOVJ C00858 BC00858 VJ=100.00  +MOVJ EC00858 VJ=100.00
MOVJ C00859 BC00859 VJ=100.00  +MOVJ EC00859 VJ=100.00
MOVL C00860 BC00860 V=666.7  +MOVJ EC00860 VJ=100.00
SMOVL C00861 BC00861 V=166.7  +MOVJ EC00861
SREFP 3 C00862 BC00862  +REFP EC00862
CALL JOB:SEARCH-R1-S13D
SET P073 P006
SFTON3D P073
SMOVL C00863 BC00863 V=166.7  +MOVJ EC00863
SMOVL C00864 BC00864 V=166.7  +MOVJ EC00864
SREFP 3 C00865 BC00865  +REFP EC00865
CALL JOB:SEARCH-R1-S13D
SET P073 P006
SFTON3D P073
SMOVL C00866 BC00866 V=166.7  +MOVJ EC00866
SMOVL C00867 BC00867 V=166.7  +MOVJ EC00867
SREFP 3 C00868 BC00868  +REFP EC00868
CALL JOB:SEARCH-R1-S13D
SET P073 P006
SFTON3D P073
SMOVL C00869 BC00869 V=166.7  +MOVJ EC00869
MOVL C00870 BC00870 V=1000.0  +MOVJ EC00870 VJ=100.00
'EndPath S4857
MOVJ C00871 BC00871 VJ=100.00  +MOVJ EC00871 VJ=100.00
MOVJ C00872 BC00872 VJ=100.00  +MOVJ EC00872 VJ=100.00
'Path S4858
SFTOF3D
MOVJ C00873 BC00873 VJ=100.00  +MOVJ EC00873 VJ=100.00
MOVL C00874 BC00874 V=666.7  +MOVJ EC00874 VJ=100.00
SMOVL C00875 BC00875 V=166.7  +MOVJ EC00875
SREFP 3 C00876 BC00876  +REFP EC00876
CALL JOB:SEARCH-R1-S13D
SET P074 P006
SFTON3D P074
SMOVL C00877 BC00877 V=166.7  +MOVJ EC00877
SREFP 3 C00878 BC00878  +REFP EC00878
CALL JOB:SEARCH-R1-S13D
SET P074 P006
SFTON3D P074
SMOVL C00879 BC00879 V=166.7  +MOVJ EC00879
MOVL C00880 BC00880 V=1000.0  +MOVJ EC00880 VJ=100.00
'EndPath S4858
MOVJ C00881 BC00881 VJ=100.00  +MOVJ EC00881 VJ=100.00
MOVJ C00882 BC00882 VJ=100.00  +MOVJ EC00882 VJ=100.00
'Path S4100
SFTOF3D
MOVJ C00883 BC00883 VJ=100.00  +MOVJ EC00883 VJ=100.00
MOVL C00884 BC00884 V=666.7  +MOVJ EC00884 VJ=100.00
SMOVL C00885 BC00885 V=166.7  +MOVJ EC00885
SREFP 3 C00886 BC00886  +REFP EC00886
CALL JOB:SEARCH-R1-S13D
SET P081 P006
SFTON3D P081
SMOVL C00887 BC00887 V=166.7  +MOVJ EC00887
SREFP 3 C00888 BC00888  +REFP EC00888
CALL JOB:SEARCH-R1-S13D
SET P081 P006
SFTON3D P081
SMOVL C00889 BC00889 V=166.7  +MOVJ EC00889
SMOVL C00890 BC00890 V=666.7  +MOVJ EC00890
SMOVL C00891 BC00891 V=666.7  +MOVJ EC00891
SMOVL C00892 BC00892 V=666.7  +MOVJ EC00892
SMOVL C00893 BC00893 V=166.7  +MOVJ EC00893
SREFP 3 C00894 BC00894  +REFP EC00894
CALL JOB:SEARCH-R1-S13D
SET P081 P006
SFTON3D P081
SMOVL C00895 BC00895 V=250.0  +MOVJ EC00895
SMOVL C00896 BC00896 V=666.7  +MOVJ EC00896
MOVJ C00897 BC00897 VJ=100.00  +MOVJ EC00897 VJ=100.00
MOVL C00898 BC00898 V=666.7  +MOVJ EC00898 VJ=100.00
SMOVL C00899 BC00899 V=166.7  +MOVJ EC00899
SREFP 3 C00900 BC00900  +REFP EC00900
CALL JOB:SEARCH-R1-S13D
SET P026 P006
SFTON3D P026
SMOVL C00901 BC00901 V=166.7  +MOVJ EC00901
SREFP 3 C00902 BC00902  +REFP EC00902
CALL JOB:SEARCH-R1-S13D
SET P026 P006
SFTON3D P026
SMOVL C00903 BC00903 V=166.7  +MOVJ EC00903
SMOVL C00904 BC00904 V=666.7  +MOVJ EC00904
SMOVL C00905 BC00905 V=666.7  +MOVJ EC00905
SMOVL C00906 BC00906 V=666.7  +MOVJ EC00906
SMOVL C00907 BC00907 V=166.7  +MOVJ EC00907
SREFP 3 C00908 BC00908  +REFP EC00908
CALL JOB:SEARCH-R1-S13D
SET P026 P006
SFTON3D P026
SMOVL C00909 BC00909 V=250.0  +MOVJ EC00909
SMOVL C00910 BC00910 V=666.7  +MOVJ EC00910
MOVL C00911 BC00911 V=1000.0  +MOVJ EC00911 VJ=100.00
'EndPath S4100
MOVJ C00912 BC00912 VJ=50.00  +MOVJ EC00912 VJ=100.00
'Path S4101
SFTOF3D
MOVJ C00913 BC00913 VJ=50.00  +MOVJ EC00913 VJ=100.00
MOVL C00914 BC00914 V=666.7  +MOVJ EC00914 VJ=100.00
SMOVL C00915 BC00915 V=166.7  +MOVJ EC00915
SREFP 3 C00916 BC00916  +REFP EC00916
CALL JOB:SEARCH-R1-S13D
SET P025 P006
SFTON3D P025
SMOVL C00917 BC00917 V=166.7  +MOVJ EC00917
SREFP 3 C00918 BC00918  +REFP EC00918
CALL JOB:SEARCH-R1-S13D
SET P025 P006
SFTON3D P025
SMOVL C00919 BC00919 V=166.7  +MOVJ EC00919
SMOVL C00920 BC00920 V=333.3  +MOVJ EC00920
SMOVL C00921 BC00921 V=166.7  +MOVJ EC00921
SREFP 3 C00922 BC00922  +REFP EC00922
CALL JOB:SEARCH-R1-S13D
SET P025 P006
SFTON3D P025
SMOVL C00923 BC00923 V=166.7  +MOVJ EC00923
MOVL C00924 BC00924 V=1000.0  +MOVJ EC00924 VJ=100.00
'EndPath S4101
MOVJ C00925 BC00925 VJ=100.00  +MOVJ EC00925 VJ=100.00
'Path S4102
SFTOF3D
MOVJ C00926 BC00926 VJ=100.00  +MOVJ EC00926 VJ=100.00
MOVL C00927 BC00927 V=666.7  +MOVJ EC00927 VJ=100.00
SMOVL C00928 BC00928 V=166.7  +MOVJ EC00928
SREFP 3 C00929 BC00929  +REFP EC00929
CALL JOB:SEARCH-R1-S13D
SET P028 P006
SFTON3D P028
SMOVL C00930 BC00930 V=166.7  +MOVJ EC00930
SREFP 3 C00931 BC00931  +REFP EC00931
CALL JOB:SEARCH-R1-S13D
SET P028 P006
SFTON3D P028
SMOVL C00932 BC00932 V=166.7  +MOVJ EC00932
SMOVL C00933 BC00933 V=333.3  +MOVJ EC00933
SMOVL C00934 BC00934 V=166.7  +MOVJ EC00934
SREFP 3 C00935 BC00935  +REFP EC00935
CALL JOB:SEARCH-R1-S13D
SET P028 P006
SFTON3D P028
SMOVL C00936 BC00936 V=166.7  +MOVJ EC00936
MOVL C00937 BC00937 V=1000.0  +MOVJ EC00937 VJ=100.00
'EndPath S4102
MOVJ C00938 BC00938 VJ=100.00  +MOVJ EC00938 VJ=100.00
'Path S4103
SFTOF3D
MOVJ C00939 BC00939 VJ=100.00  +MOVJ EC00939 VJ=100.00
MOVL C00940 BC00940 V=666.7  +MOVJ EC00940 VJ=100.00
SMOVL C00941 BC00941 V=166.7  +MOVJ EC00941
SREFP 3 C00942 BC00942  +REFP EC00942
CALL JOB:SEARCH-R1-S13D
SET P033 P006
SFTON3D P033
SMOVL C00943 BC00943 V=166.7  +MOVJ EC00943
SMOVL C00944 BC00944 V=166.7  +MOVJ EC00944
SREFP 3 C00945 BC00945  +REFP EC00945
CALL JOB:SEARCH-R1-S13D
SET P033 P006
SFTON3D P033
SMOVL C00946 BC00946 V=166.7  +MOVJ EC00946
SMOVL C00947 BC00947 V=166.7  +MOVJ EC00947
SMOVL C00948 BC00948 V=166.7  +MOVJ EC00948
SREFP 3 C00949 BC00949  +REFP EC00949
CALL JOB:SEARCH-R1-S13D
SET P033 P006
SFTON3D P033
SMOVL C00950 BC00950 V=166.7  +MOVJ EC00950
MOVL C00951 BC00951 V=1000.0  +MOVJ EC00951 VJ=100.00
'EndPath S4103
'Path S4104
SFTOF3D
MOVJ C00952 BC00952 VJ=100.00  +MOVJ EC00952 VJ=100.00
MOVL C00953 BC00953 V=666.7  +MOVJ EC00953 VJ=100.00
SMOVL C00954 BC00954 V=166.7  +MOVJ EC00954
SREFP 3 C00955 BC00955  +REFP EC00955
CALL JOB:SEARCH-R1-S13D
SET P027 P006
SFTON3D P027
SMOVL C00956 BC00956 V=250.0  +MOVJ EC00956
SMOVL C00957 BC00957 V=166.7  +MOVJ EC00957
SREFP 3 C00958 BC00958  +REFP EC00958
CALL JOB:SEARCH-R1-S13D
SET P027 P006
SFTON3D P027
SMOVL C00959 BC00959 V=166.7  +MOVJ EC00959
SMOVL C00960 BC00960 V=166.7  +MOVJ EC00960
SREFP 3 C00961 BC00961  +REFP EC00961
CALL JOB:SEARCH-R1-S13D
SET P027 P006
SFTON3D P027
SMOVL C00962 BC00962 V=166.7  +MOVJ EC00962
MOVL C00963 BC00963 V=1000.0  +MOVJ EC00963 VJ=100.00
'EndPath S4104
MOVJ C00964 BC00964 VJ=100.00  +MOVJ EC00964 VJ=100.00
'Path S4105
SFTOF3D
MOVJ C00965 BC00965 VJ=100.00  +MOVJ EC00965 VJ=100.00
MOVL C00966 BC00966 V=666.7  +MOVJ EC00966 VJ=100.00
SMOVL C00967 BC00967 V=166.7  +MOVJ EC00967
SREFP 3 C00968 BC00968  +REFP EC00968
CALL JOB:SEARCH-R1-S13D
SET P030 P006
SFTON3D P030
SMOVL C00969 BC00969 V=166.7  +MOVJ EC00969
SREFP 3 C00970 BC00970  +REFP EC00970
CALL JOB:SEARCH-R1-S13D
SET P030 P006
SFTON3D P030
SMOVL C00971 BC00971 V=166.7  +MOVJ EC00971
MOVL C00972 BC00972 V=1000.0  +MOVJ EC00972 VJ=100.00
'EndPath S4105
'Path S4106
SFTOF3D
MOVJ C00973 BC00973 VJ=100.00  +MOVJ EC00973 VJ=100.00
MOVL C00974 BC00974 V=666.7  +MOVJ EC00974 VJ=100.00
SMOVL C00975 BC00975 V=166.7  +MOVJ EC00975
SREFP 3 C00976 BC00976  +REFP EC00976
CALL JOB:SEARCH-R1-S13D
SET P031 P006
SFTON3D P031
SMOVL C00977 BC00977 V=166.7  +MOVJ EC00977
SREFP 3 C00978 BC00978  +REFP EC00978
CALL JOB:SEARCH-R1-S13D
SET P031 P006
SFTON3D P031
SMOVL C00979 BC00979 V=166.7  +MOVJ EC00979
SFTOF3D
MOVL C00980 BC00980 V=666.7  +MOVJ EC00980 VJ=100.00
SMOVL C00981 BC00981 V=166.7  +MOVJ EC00981
SREFP 3 C00982 BC00982  +REFP EC00982
CALL JOB:SEARCH-R1-S13D
SET P098 P006
SFTON3D P098
SMOVL C00983 BC00983 V=166.7  +MOVJ EC00983
SREFP 3 C00984 BC00984  +REFP EC00984
CALL JOB:SEARCH-R1-S13D
SET P098 P006
SFTON3D P098
SMOVL C00985 BC00985 V=166.7  +MOVJ EC00985
MOVL C00986 BC00986 V=1000.0  +MOVJ EC00986 VJ=100.00
'EndPath S4106
MOVJ C00987 BC00987 VJ=100.00  +MOVJ EC00987 VJ=100.00
'Path S4107
SFTOF3D
MOVJ C00988 BC00988 VJ=100.00  +MOVJ EC00988 VJ=100.00
MOVL C00989 BC00989 V=666.7  +MOVJ EC00989 VJ=100.00
SMOVL C00990 BC00990 V=166.7  +MOVJ EC00990
SREFP 3 C00991 BC00991  +REFP EC00991
CALL JOB:SEARCH-R1-S13D
SET P032 P006
SFTON3D P032
SMOVL C00992 BC00992 V=166.7  +MOVJ EC00992
SREFP 3 C00993 BC00993  +REFP EC00993
CALL JOB:SEARCH-R1-S13D
SET P032 P006
SFTON3D P032
SMOVL C00994 BC00994 V=166.7  +MOVJ EC00994
SMOVL C00995 BC00995 V=250.0  +MOVJ EC00995
SMOVL C00996 BC00996 V=166.7  +MOVJ EC00996
SREFP 3 C00997 BC00997  +REFP EC00997
CALL JOB:SEARCH-R1-S13D
SET P032 P006
SFTON3D P032
SMOVL C00998 BC00998 V=166.7  +MOVJ EC00998
MOVL C00999 BC00999 V=1000.0  +MOVJ EC00999 VJ=100.00
'EndPath S4107
'
MOVJ C01000 BC01000 VJ=100.00  +MOVJ EC01000 VJ=100.00
'Path S4208
SFTOF3D
MOVJ C01001 BC01001 VJ=100.00  +MOVJ EC01001 VJ=100.00
MOVL C01002 BC01002 V=666.7  +MOVJ EC01002 VJ=100.00
SMOVL C01003 BC01003 V=166.7  +MOVJ EC01003
SREFP 3 C01004 BC01004  +REFP EC01004
CALL JOB:SEARCH-R1-S13D
SET P052 P006
SFTON3D P052
SMOVL C01005 BC01005 V=166.7  +MOVJ EC01005
SREFP 3 C01006 BC01006  +REFP EC01006
CALL JOB:SEARCH-R1-S13D
SET P052 P006
SFTON3D P052
SMOVL C01007 BC01007 V=166.7  +MOVJ EC01007
SFTOF3D
MOVL C01008 BC01008 V=1000.0  +MOVJ EC01008 VJ=100.00
SMOVL C01009 BC01009 V=500.0  +MOVJ EC01009
SMOVL C01010 BC01010 V=166.7  +MOVJ EC01010
SREFP 3 C01011 BC01011  +REFP EC01011
CALL JOB:SEARCH-R1-S13D
SET P088 P006
SFTON3D P088
SMOVL C01012 BC01012 V=166.7  +MOVJ EC01012
SMOVL C01013 BC01013 V=166.7  +MOVJ EC01013
SMOVL C01014 BC01014 V=166.7  +MOVJ EC01014
SREFP 3 C01015 BC01015  +REFP EC01015
CALL JOB:SEARCH-R1-S13D
SET P088 P006
SFTON3D P088
SMOVL C01016 BC01016 V=333.3  +MOVJ EC01016
SMOVL C01017 BC01017 V=666.7  +MOVJ EC01017
SFTOF3D
'EndPath S4208
MOVJ C01018 BC01018 VJ=100.00  +MOVJ EC01018 VJ=100.00
'Path S4209
SFTOF3D
MOVJ C01019 BC01019 VJ=100.00  +MOVJ EC01019 VJ=100.00
MOVL C01020 BC01020 V=666.7  +MOVJ EC01020 VJ=100.00
SMOVL C01021 BC01021 V=166.7  +MOVJ EC01021
SREFP 3 C01022 BC01022  +REFP EC01022
CALL JOB:SEARCH-R1-S13D
SET P053 P006
SFTON3D P053
SMOVL C01023 BC01023 V=166.7  +MOVJ EC01023
SMOVL C01024 BC01024 V=166.7  +MOVJ EC01024
SREFP 3 C01025 BC01025  +REFP EC01025
CALL JOB:SEARCH-R1-S13D
SET P053 P006
SFTON3D P053
SMOVL C01026 BC01026 V=166.7  +MOVJ EC01026
MOVL C01027 BC01027 V=1000.0  +MOVJ EC01027 VJ=100.00
'EndPath S4209
*BP1
MOVJ C01028 BC01028 VJ=100.00  +MOVJ EC01028 VJ=100.00
'Path W4108
SFTOF3D
SFTON3D P033
MOVJ C01029 BC01029 VJ=100.00  +MOVJ EC01029 VJ=100.00
SMOVL C01030 BC01030 V=666.7  +MOVJ EC01030
SMOVL C01031 BC01031 V=166.7 PL=0  +MOVJ EC01031
MACRO1 MJ#(0) ARGF14
ARCON
SMOVL C01032 BC01032 V=9.2  +MOVJ EC01032
ARCOF
SMOVL C01033 BC01033 V=800.0  +MOVJ EC01033
SMOVL C01034 BC01034 V=1000.0  +MOVJ EC01034
SFTOF3D
'EndPath W4108
'Path W4109
SFTOF3D
MOVJ C01035 BC01035 VJ=100.00  +MOVJ EC01035 VJ=100.00
MOVJ C01036 BC01036 VJ=100.00  +MOVJ EC01036 VJ=100.00
'Path W4110
SFTOF3D
SFTON3D P033
MOVJ C01037 BC01037 VJ=100.00  +MOVJ EC01037 VJ=100.00
SMOVL C01038 BC01038 V=800.0  +MOVJ EC01038
SMOVL C01039 BC01039 V=133.3 PL=0  +MOVJ EC01039
MACRO1 MJ#(0) ARGF9
ARCON
SMOVL C01040 BC01040 V=11.7  +MOVJ EC01040
SMOVL C01041 BC01041 V=11.7  +MOVJ EC01041
SMOVL C01042 BC01042 V=11.7  +MOVJ EC01042
ARCOF
SMOVL C01043 BC01043 V=800.0  +MOVJ EC01043
SMOVL C01044 BC01044 V=1000.0  +MOVJ EC01044
SFTOF3D
'EndPath W4110
MOVJ C01045 BC01045 VJ=100.00  +MOVJ EC01045 VJ=100.00
'9
MOVJ C01046 BC01046 VJ=100.00  +MOVJ EC01046 VJ=100.00
'Path W4111
SFTOF3D
SFTON3D P026
MOVJ C01047 BC01047 VJ=100.00  +MOVJ EC01047 VJ=100.00
SMOVL C01048 BC01048 V=666.7  +MOVJ EC01048
SMOVL C01049 BC01049 V=166.7 PL=0  +MOVJ EC01049
MACRO1 MJ#(0) ARGF14
ARCON
SMOVL C01050 BC01050 V=9.2  +MOVJ EC01050
ARCOF
SMOVL C01051 BC01051 V=800.0  +MOVJ EC01051
SMOVL C01052 BC01052 V=1000.0  +MOVJ EC01052
SFTOF3D
'EndPath W4111
'Path W4112
SFTOF3D
SFTON3D P026
MOVJ C01053 BC01053 VJ=100.00  +MOVJ EC01053 VJ=100.00
SMOVL C01054 BC01054 V=800.0  +MOVJ EC01054
SMOVL C01055 BC01055 V=150.0 PL=0  +MOVJ EC01055
ARCON
SMOVL C01056 BC01056 V=11.7  +MOVJ EC01056
SMOVL C01057 BC01057 V=11.7  +MOVJ EC01057
SMOVL C01058 BC01058 V=11.7  +MOVJ EC01058
ARCOF
SMOVL C01059 BC01059 V=800.0  +MOVJ EC01059
SMOVL C01060 BC01060 V=1000.0  +MOVJ EC01060
SFTOF3D
MOVJ C01061 BC01061 VJ=100.00  +MOVJ EC01061 VJ=100.00
MOVJ C01062 BC01062 VJ=100.00  +MOVJ EC01062 VJ=100.00
'uwaga na podajnik
'Path W4114
SFTOF3D
SFTON3D P026
MOVJ C01063 BC01063 VJ=100.00  +MOVJ EC01063 VJ=100.00
SMOVL C01064 BC01064 V=800.0  +MOVJ EC01064
SMOVL C01065 BC01065 V=150.0 PL=0  +MOVJ EC01065
ARCON
SMOVL C01066 BC01066 V=11.7  +MOVJ EC01066
ARCOF
SMOVL C01067 BC01067 V=800.0  +MOVJ EC01067
SMOVL C01068 BC01068 V=1000.0  +MOVJ EC01068
SFTOF3D
'EndPath W4114
'brak dostepu offset drutu 1cm
'Path W4115
SFTOF3D
SFTON3D P026
MOVJ C01069 BC01069 VJ=100.00  +MOVJ EC01069 VJ=100.00
SMOVL C01070 BC01070 V=800.0  +MOVJ EC01070
SMOVL C01071 BC01071 V=150.0 PL=0  +MOVJ EC01071
ARCON
SMOVL C01072 BC01072 V=11.7  +MOVJ EC01072
ARCOF
SMOVL C01073 BC01073 V=800.0  +MOVJ EC01073
SMOVL C01074 BC01074 V=1000.0  +MOVJ EC01074
SFTOF3D
SFTON3D P081
MOVJ C01075 BC01075 VJ=100.00  +MOVJ EC01075 VJ=100.00
SMOVL C01076 BC01076 V=666.7  +MOVJ EC01076
SMOVL C01077 BC01077 V=166.7 PL=0  +MOVJ EC01077
MACRO1 MJ#(0) ARGF14
ARCON
SMOVL C01078 BC01078 V=9.2  +MOVJ EC01078
ARCOF
SMOVL C01079 BC01079 V=800.0  +MOVJ EC01079
SMOVL C01080 BC01080 V=1000.0  +MOVJ EC01080
SFTOF3D
'EndPath W4111
'Path W4112
SFTOF3D
SFTON3D P081
MOVJ C01081 BC01081 VJ=100.00  +MOVJ EC01081 VJ=100.00
SMOVL C01082 BC01082 V=800.0  +MOVJ EC01082
SMOVL C01083 BC01083 V=150.0 PL=0  +MOVJ EC01083
ARCON
SMOVL C01084 BC01084 V=11.7  +MOVJ EC01084
SMOVL C01085 BC01085 V=11.7  +MOVJ EC01085
SMOVL C01086 BC01086 V=11.7  +MOVJ EC01086
ARCOF
SMOVL C01087 BC01087 V=800.0  +MOVJ EC01087
SMOVL C01088 BC01088 V=1000.0  +MOVJ EC01088
SFTOF3D
MOVJ C01089 BC01089 VJ=100.00  +MOVJ EC01089 VJ=100.00
MOVJ C01090 BC01090 VJ=100.00  +MOVJ EC01090 VJ=100.00
'uwaga na podajnik
'Path W4114
SFTOF3D
SFTON3D P081
MOVJ C01091 BC01091 VJ=100.00  +MOVJ EC01091 VJ=100.00
SMOVL C01092 BC01092 V=800.0  +MOVJ EC01092
SMOVL C01093 BC01093 V=150.0 PL=0  +MOVJ EC01093
ARCON
SMOVL C01094 BC01094 V=11.7  +MOVJ EC01094
ARCOF
SMOVL C01095 BC01095 V=800.0  +MOVJ EC01095
SMOVL C01096 BC01096 V=1000.0  +MOVJ EC01096
SFTOF3D
'EndPath W4114
'brak dostepu offset drutu 1cm
'Path W4115
SFTOF3D
SFTON3D P081
MOVJ C01097 BC01097 VJ=100.00  +MOVJ EC01097 VJ=100.00
SMOVL C01098 BC01098 V=800.0  +MOVJ EC01098
SMOVL C01099 BC01099 V=150.0 PL=0  +MOVJ EC01099
ARCON
SMOVL C01100 BC01100 V=11.7  +MOVJ EC01100
ARCOF
SMOVL C01101 BC01101 V=800.0  +MOVJ EC01101
SMOVL C01102 BC01102 V=1000.0  +MOVJ EC01102
SFTOF3D
'EndPath W4115
MOVJ C01103 BC01103 VJ=100.00  +MOVJ EC01103 VJ=100.00
'10
'11
MOVJ C01104 BC01104 VJ=100.00  +MOVJ EC01104 VJ=100.00
'Path W4118
SFTOF3D
SFTON3D P025
MOVJ C01105 BC01105 VJ=100.00  +MOVJ EC01105 VJ=100.00
SMOVL C01106 BC01106 V=800.0  +MOVJ EC01106
SMOVL C01107 BC01107 V=166.7  +MOVJ EC01107
ARCON
SMOVL C01108 BC01108 V=9.2  +MOVJ EC01108
SMOVL C01109 BC01109 V=9.2  +MOVJ EC01109
SMOVL C01110 BC01110 V=9.2  +MOVJ EC01110
SMOVL C01111 BC01111 V=9.2  +MOVJ EC01111
SMOVL C01112 BC01112 V=9.2  +MOVJ EC01112
ARCOF
SMOVL C01113 BC01113 V=800.0  +MOVJ EC01113
SMOVL C01114 BC01114 V=1000.0  +MOVJ EC01114
SFTOF3D
'EndPath W4118
'brak dostepu offset drutu 1cm
MOVJ C01115 BC01115 VJ=100.00  +MOVJ EC01115 VJ=100.00
'Path W4117
SFTOF3D
SFTON3D P025
MOVJ C01116 BC01116 VJ=100.00  +MOVJ EC01116 VJ=100.00
SMOVL C01117 BC01117 V=800.0  +MOVJ EC01117
SMOVL C01118 BC01118 V=166.7 PL=0  +MOVJ EC01118
ARCON
SMOVL C01119 BC01119 V=10.0  +MOVJ EC01119
ARCOF
SMOVL C01120 BC01120 V=800.0  +MOVJ EC01120
SMOVL C01121 BC01121 V=1000.0  +MOVJ EC01121
SFTOF3D
'EndPath W4117
'12
MOVJ C01122 BC01122 VJ=100.00  +MOVJ EC01122 VJ=100.00
MOVJ C01123 BC01123 VJ=100.00  +MOVJ EC01123 VJ=100.00
'Path W4859
SFTOF3D
SFTON3D P073
MOVJ C01124 BC01124 VJ=100.00  +MOVJ EC01124 VJ=100.00
SMOVL C01125 BC01125 V=800.0  +MOVJ EC01125
SMOVL C01126 BC01126 V=150.0 PL=0  +MOVJ EC01126
ARCON
SMOVL C01127 BC01127 V=8.3  +MOVJ EC01127
SFTON3D P074
SMOVL C01128 BC01128 V=9.2  +MOVJ EC01128
ARCOF
SMOVL C01129 BC01129 V=333.3  +MOVJ EC01129
SMOVL C01130 BC01130 V=333.3  +MOVJ EC01130
SMOVL C01131 BC01131 V=333.3  +MOVJ EC01131
SMOVL C01132 BC01132 V=166.7 PL=0  +MOVJ EC01132
ARCON
SMOVL C01133 BC01133 V=9.2  +MOVJ EC01133
SMOVL C01134 BC01134 V=9.2  +MOVJ EC01134
ARCOF
SMOVL C01135 BC01135 V=800.0  +MOVJ EC01135
SMOVL C01136 BC01136 V=1000.0  +MOVJ EC01136
SFTOF3D
'EndPath W4859
MOVJ C01137 BC01137 VJ=100.00  +MOVJ EC01137 VJ=100.00
MOVJ C01138 BC01138 VJ=100.00  +MOVJ EC01138 VJ=100.00
'Path W4119
SFTOF3D
SFTON3D P034
MOVJ C01139 BC01139 VJ=100.00  +MOVJ EC01139 VJ=100.00
SMOVL C01140 BC01140 V=800.0  +MOVJ EC01140
SMOVL C01141 BC01141 V=150.0 PL=0  +MOVJ EC01141
ARCON
SMOVL C01142 BC01142 V=10.0  +MOVJ EC01142
SMOVL C01143 BC01143 V=10.0  +MOVJ EC01143
SMOVL C01144 BC01144 V=10.0  +MOVJ EC01144
ARCOF
SMOVL C01145 BC01145 V=800.0  +MOVJ EC01145
SMOVL C01146 BC01146 V=1000.0  +MOVJ EC01146
SFTOF3D
'EndPath W4119
'Path W4210
SFTOF3D
SFTON3D P050
MOVJ C01147 BC01147 VJ=100.00  +MOVJ EC01147 VJ=100.00
SMOVL C01148 BC01148 V=800.0  +MOVJ EC01148
SMOVL C01149 BC01149 V=150.0 PL=0  +MOVJ EC01149
ARCON
SMOVL C01150 BC01150 V=11.7  +MOVJ EC01150
ARCOF
SMOVL C01151 BC01151 V=800.0  +MOVJ EC01151
SMOVL C01152 BC01152 V=1000.0  +MOVJ EC01152
SFTOF3D
'EndPath W4210
'Path W4211
SFTOF3D
SFTON3D P034
MOVJ C01153 BC01153 VJ=100.00  +MOVJ EC01153 VJ=100.00
SMOVL C01154 BC01154 V=800.0  +MOVJ EC01154
SMOVL C01155 BC01155 V=166.7 PL=0  +MOVJ EC01155
ARCON
SWVON WEV#(66)
SMOVL C01156 BC01156 V=9.2  +MOVJ EC01156
SMOVL C01157 BC01157 V=9.2  +MOVJ EC01157
SMOVL C01158 BC01158 V=9.2  +MOVJ EC01158
ARCOF
SWVOF
SMOVL C01159 BC01159 V=800.0  +MOVJ EC01159
SMOVL C01160 BC01160 V=1000.0  +MOVJ EC01160
MOVJ C01161 BC01161 VJ=30.00  +MOVJ EC01161 VJ=30.00
MOVJ C01162 BC01162 VJ=30.00  +MOVJ EC01162 VJ=30.00
SFTOF3D
MACRO1 MJ#(0) ARGF6
MOVJ C01163 BC01163 VJ=30.00  +MOVJ EC01163 VJ=30.00
SFTON3D P063
SMOVL C01164 BC01164 V=133.3  +MOVJ EC01164
ARCON
SMOVL C01165 BC01165 V=11.7  +MOVJ EC01165
SMOVL C01166 BC01166 V=11.7  +MOVJ EC01166
SMOVL C01167 BC01167 V=11.7  +MOVJ EC01167
SFTON3D P062
SMOVL C01168 BC01168 V=11.7  +MOVJ EC01168
SMOVL C01169 BC01169 V=11.7  +MOVJ EC01169
SFTON3D P061
SMOVL C01170 BC01170 V=11.0  +MOVJ EC01170
SMOVL C01171 BC01171 V=11.0  +MOVJ EC01171
ARCOF
SMOVL C01172 BC01172 V=250.0  +MOVJ EC01172
SFTOF3D
MOVJ C01173 BC01173 VJ=30.00  +MOVJ EC01173 VJ=30.00
MOVJ C01174 BC01174 VJ=30.00  +MOVJ EC01174 VJ=30.00
'EndPath W4211
'Path W4210
SFTOF3D
SFTON3D P054
MOVJ C01175 BC01175 VJ=100.00  +MOVJ EC01175 VJ=100.00
SMOVL C01176 BC01176 V=800.0  +MOVJ EC01176
SMOVL C01177 BC01177 V=150.0 PL=0  +MOVJ EC01177
MACRO1 MJ#(0) ARGF14
ARCON
SWVON WEV#(67)
SMOVL C01178 BC01178 V=10.0  +MOVJ EC01178
SMOVL C01179 BC01179 V=10.0  +MOVJ EC01179
ARCOF
SWVOF
SMOVL C01180 BC01180 V=800.0  +MOVJ EC01180
SMOVL C01181 BC01181 V=1000.0  +MOVJ EC01181
SFTOF3D
'EndPath W4210
'Path W4121
SFTOF3D
SFTON3D P028
MOVJ C01182 BC01182 VJ=100.00  +MOVJ EC01182 VJ=100.00
SMOVL C01183 BC01183 V=800.0  +MOVJ EC01183
SMOVL C01184 BC01184 V=150.0 PL=0  +MOVJ EC01184
ARCON
SMOVL C01185 BC01185 V=9.2  +MOVJ EC01185
SMOVL C01186 BC01186 V=9.2  +MOVJ EC01186
SMOVL C01187 BC01187 V=9.2  +MOVJ EC01187
ARCOF
SMOVL C01188 BC01188 V=800.0  +MOVJ EC01188
SMOVL C01189 BC01189 V=1000.0  +MOVJ EC01189
SFTOF3D
'EndPath W4121
'brak dostepu offset 5mm
MOVJ C01190 BC01190 VJ=100.00  +MOVJ EC01190 VJ=100.00
'Path W4122
SFTOF3D
SFTON3D P028
MOVJ C01191 BC01191 VJ=100.00  +MOVJ EC01191 VJ=100.00
SMOVL C01192 BC01192 V=800.0  +MOVJ EC01192
SMOVL C01193 BC01193 V=166.7 PL=0  +MOVJ EC01193
ARCON
SMOVL C01194 BC01194 V=11.7  +MOVJ EC01194
ARCOF
SMOVL C01195 BC01195 V=800.0  +MOVJ EC01195
SMOVL C01196 BC01196 V=1000.0  +MOVJ EC01196
SFTOF3D
'EndPath W4122
MOVJ C01197 BC01197 VJ=100.00  +MOVJ EC01197 VJ=100.00
'13
MOVJ C01198 BC01198 VJ=100.00  +MOVJ EC01198 VJ=100.00
'Path W4123
SFTOF3D
SFTON3D P030
MOVJ C01199 BC01199 VJ=100.00  +MOVJ EC01199 VJ=100.00
SMOVL C01200 BC01200 V=800.0  +MOVJ EC01200
SMOVL C01201 BC01201 V=150.0 PL=0  +MOVJ EC01201
SREFP 1 C01202 BC01202  +REFP EC01202
SREFP 2 C01203 BC01203  +REFP EC01203
MACRO1 MJ#(0) ARGF9
ARCON
SWVON WEV#(10)
SFTON3D P031
SMOVL C01204 BC01204 V=9.2  +MOVJ EC01204
SFTON3D P098
SMOVL C01205 BC01205 V=9.2  +MOVJ EC01205
SMOVL C01206 BC01206 V=9.2  +MOVJ EC01206
ARCOF
SWVOF
SMOVL C01207 BC01207 V=800.0  +MOVJ EC01207
SMOVL C01208 BC01208 V=1000.0  +MOVJ EC01208
SFTOF3D
'EndPath W4123
'14
'15-brak
'Path W4212
SFTOF3D
SFTON3D P052
MOVJ C01209 BC01209 VJ=100.00  +MOVJ EC01209 VJ=100.00
SMOVL C01210 BC01210 V=800.0  +MOVJ EC01210
SMOVL C01211 BC01211 V=150.0 PL=0  +MOVJ EC01211
ARCON
SMOVL C01212 BC01212 V=10.8  +MOVJ EC01212
SMOVL C01213 BC01213 V=10.8  +MOVJ EC01213
SMOVL C01214 BC01214 V=10.8  +MOVJ EC01214
ARCOF
SMOVL C01215 BC01215 V=800.0  +MOVJ EC01215
MACRO1 MJ#(0) ARGF6
SMOVL C01216 BC01216 V=333.3  +MOVJ EC01216
SFTOF3D
'DODAC SHIFT
SFTON3D P088
SMOVL C01217 BC01217 V=133.3  +MOVJ EC01217
ARCON
SMOVL C01218 BC01218 V=10.8  +MOVJ EC01218
ARCOF
SMOVL C01219 BC01219 V=250.0  +MOVJ EC01219
SMOVL C01220 BC01220 V=1000.0  +MOVJ EC01220
SFTOF3D
'EndPath W4212
'16
'Path W4213
SFTOF3D
SFTON3D P053
MOVJ C01221 BC01221 VJ=100.00  +MOVJ EC01221 VJ=100.00
SMOVL C01222 BC01222 V=800.0  +MOVJ EC01222
SMOVL C01223 BC01223 V=150.0 PL=0  +MOVJ EC01223
MACRO1 MJ#(0) ARGF9
ARCON
SMOVL C01224 BC01224 V=10.8  +MOVJ EC01224
SMOVL C01225 BC01225 V=10.8  +MOVJ EC01225
SMOVL C01226 BC01226 V=10.8  +MOVJ EC01226
ARCOF
SMOVL C01227 BC01227 V=800.0  +MOVJ EC01227
SMOVL C01228 BC01228 V=1000.0  +MOVJ EC01228
SFTOF3D
'EndPath W4213
'Path W4124
SFTOF3D
SFTON3D P029
MOVJ C01229 BC01229 VJ=100.00  +MOVJ EC01229 VJ=100.00
SMOVL C01230 BC01230 V=800.0  +MOVJ EC01230
SMOVL C01231 BC01231 V=166.7 PL=0  +MOVJ EC01231
MACRO1 MJ#(0) ARGF14
COMM ARCON
SMOVL C01232 BC01232 V=10.0  +MOVJ EC01232
SMOVL C01233 BC01233 V=10.0  +MOVJ EC01233
ARCOF
SMOVL C01234 BC01234 V=800.0  +MOVJ EC01234
SMOVL C01235 BC01235 V=1000.0  +MOVJ EC01235
SFTOF3D
'EndPath W4124
MOVJ C01236 BC01236 VJ=100.00  +MOVJ EC01236 VJ=100.00
'Path W4125
SFTOF3D
SFTON3D P029
MOVJ C01237 BC01237 VJ=100.00  +MOVJ EC01237 VJ=100.00
SMOVL C01238 BC01238 V=800.0  +MOVJ EC01238
SMOVL C01239 BC01239 V=150.0 PL=0  +MOVJ EC01239
COMM ARCON
SMOVL C01240 BC01240 V=11.7  +MOVJ EC01240
SMOVL C01241 BC01241 V=11.7  +MOVJ EC01241
SMOVL C01242 BC01242 V=11.7  +MOVJ EC01242
ARCOF
SMOVL C01243 BC01243 V=800.0  +MOVJ EC01243
SMOVL C01244 BC01244 V=1000.0  +MOVJ EC01244
SFTOF3D
'EndPath W4125
MOVJ C01245 BC01245 VJ=100.00  +MOVJ EC01245 VJ=100.00
'Path W4126
SFTOF3D
SFTON3D P029
MOVJ C01246 BC01246 VJ=100.00  +MOVJ EC01246 VJ=100.00
SMOVL C01247 BC01247 V=800.0  +MOVJ EC01247
SMOVL C01248 BC01248 V=166.7 PL=0  +MOVJ EC01248
COMM ARCON
SMOVL C01249 BC01249 V=11.7  +MOVJ EC01249
ARCON
SMOVL C01250 BC01250 V=11.7  +MOVJ EC01250
SMOVL C01251 BC01251 V=11.7  +MOVJ EC01251
ARCOF
SMOVL C01252 BC01252 V=800.0  +MOVJ EC01252
SMOVL C01253 BC01253 V=1000.0  +MOVJ EC01253
SFTOF3D
SFTON3D P080
MOVJ C01254 BC01254 VJ=100.00  +MOVJ EC01254 VJ=100.00
SMOVL C01255 BC01255 V=800.0  +MOVJ EC01255
SMOVL C01256 BC01256 V=166.7 PL=0  +MOVJ EC01256
MACRO1 MJ#(0) ARGF14
ARCON
SMOVL C01257 BC01257 V=10.0  +MOVJ EC01257
SMOVL C01258 BC01258 V=10.0  +MOVJ EC01258
ARCOF
SMOVL C01259 BC01259 V=800.0  +MOVJ EC01259
SMOVL C01260 BC01260 V=1000.0  +MOVJ EC01260
SFTOF3D
'EndPath W4124
MOVJ C01261 BC01261 VJ=100.00  +MOVJ EC01261 VJ=100.00
'Path W4125
SFTOF3D
SFTON3D P080
MOVJ C01262 BC01262 VJ=100.00  +MOVJ EC01262 VJ=100.00
SMOVL C01263 BC01263 V=800.0  +MOVJ EC01263
SMOVL C01264 BC01264 V=150.0 PL=0  +MOVJ EC01264
ARCON
SMOVL C01265 BC01265 V=11.7  +MOVJ EC01265
SMOVL C01266 BC01266 V=11.7  +MOVJ EC01266
SMOVL C01267 BC01267 V=11.7  +MOVJ EC01267
ARCOF
SMOVL C01268 BC01268 V=800.0  +MOVJ EC01268
SMOVL C01269 BC01269 V=1000.0  +MOVJ EC01269
SFTOF3D
'EndPath W4125
MOVJ C01270 BC01270 VJ=100.00  +MOVJ EC01270 VJ=100.00
'Path W4126
SFTOF3D
SFTON3D P080
MOVJ C01271 BC01271 VJ=100.00  +MOVJ EC01271 VJ=100.00
SMOVL C01272 BC01272 V=800.0  +MOVJ EC01272
SMOVL C01273 BC01273 V=166.7 PL=0  +MOVJ EC01273
ARCON
SMOVL C01274 BC01274 V=11.7  +MOVJ EC01274
ARCON
SMOVL C01275 BC01275 V=11.7  +MOVJ EC01275
SMOVL C01276 BC01276 V=11.7  +MOVJ EC01276
ARCOF
SMOVL C01277 BC01277 V=800.0  +MOVJ EC01277
SMOVL C01278 BC01278 V=1000.0  +MOVJ EC01278
SFTOF3D
'EndPath W4126
MOVJ C01279 BC01279 VJ=100.00  +MOVJ EC01279 VJ=100.00
'17
'Path W4127
SFTOF3D
SFTON3D P027
MOVJ C01280 BC01280 VJ=100.00  +MOVJ EC01280 VJ=100.00
SMOVL C01281 BC01281 V=800.0  +MOVJ EC01281
SMOVL C01282 BC01282 V=150.0 PL=0  +MOVJ EC01282
ARCON
SMOVL C01283 BC01283 V=10.0  +MOVJ EC01283
ARCOF
SMOVL C01284 BC01284 V=800.0  +MOVJ EC01284
SMOVL C01285 BC01285 V=1000.0  +MOVJ EC01285
SFTOF3D
'EndPath W4127
'Path W4128
SFTOF3D
SFTON3D P027
MOVJ C01286 BC01286 VJ=100.00  +MOVJ EC01286 VJ=100.00
SMOVL C01287 BC01287 V=800.0  +MOVJ EC01287
SMOVL C01288 BC01288 V=150.0 PL=0  +MOVJ EC01288
ARCON
SMOVL C01289 BC01289 V=11.7  +MOVJ EC01289
ARCOF
SMOVL C01290 BC01290 V=800.0  +MOVJ EC01290
SMOVL C01291 BC01291 V=1000.0  +MOVJ EC01291
SFTOF3D
'EndPath W4128
'Path W4129
SFTOF3D
SFTON3D P027
MOVJ C01292 BC01292 VJ=100.00  +MOVJ EC01292 VJ=100.00
SMOVL C01293 BC01293 V=800.0  +MOVJ EC01293
SMOVL C01294 BC01294 V=150.0 PL=0  +MOVJ EC01294
SMOVL C01295 BC01295 V=16.7  +MOVJ EC01295
ARCOF
SMOVL C01296 BC01296 V=800.0  +MOVJ EC01296
SMOVL C01297 BC01297 V=1000.0  +MOVJ EC01297
SFTOF3D
'EndPath W4129
'18
MOVJ C01298 BC01298 VJ=100.00  +MOVJ EC01298 VJ=100.00
'Path W4130
SFTOF3D
SFTON3D P024
MOVJ C01299 BC01299 VJ=100.00  +MOVJ EC01299 VJ=100.00
SMOVL C01300 BC01300 V=800.0  +MOVJ EC01300
SMOVL C01301 BC01301 V=150.0 PL=0  +MOVJ EC01301
COMM ARCON
SMOVL C01302 BC01302 V=9.2  +MOVJ EC01302
SMOVL C01303 BC01303 V=9.2  +MOVJ EC01303
SMOVL C01304 BC01304 V=9.2  +MOVJ EC01304
SMOVL C01305 BC01305 V=9.2  +MOVJ EC01305
ARCOF
SMOVL C01306 BC01306 V=800.0  +MOVJ EC01306
SMOVL C01307 BC01307 V=1000.0  +MOVJ EC01307
SFTOF3D
'EndPath W4130
'Path W4860
SFTOF3D
SFTON3D P071
MOVJ C01308 BC01308 VJ=100.00  +MOVJ EC01308 VJ=100.00
SMOVL C01309 BC01309 V=800.0  +MOVJ EC01309
SMOVL C01310 BC01310 V=150.0 PL=0  +MOVJ EC01310
MACRO1 MJ#(0) ARGF9
ARCON
SMOVL C01311 BC01311 V=9.2  +MOVJ EC01311
SFTON3D P072
ARCON
SMOVL C01312 BC01312 V=9.2  +MOVJ EC01312
SMOVL C01313 BC01313 V=9.2  +MOVJ EC01313
ARCOF
SMOVL C01314 BC01314 V=333.3  +MOVJ EC01314
SMOVL C01315 BC01315 V=666.7  +MOVJ EC01315
SMOVL C01316 BC01316 V=333.3  +MOVJ EC01316
SMOVL C01317 BC01317 V=166.7 PL=0  +MOVJ EC01317
ARCON
SMOVL C01318 BC01318 V=9.2  +MOVJ EC01318
SMOVL C01319 BC01319 V=9.2  +MOVJ EC01319
ARCOF
SMOVL C01320 BC01320 V=800.0  +MOVJ EC01320
SMOVL C01321 BC01321 V=1000.0  +MOVJ EC01321
SFTOF3D
'EndPath W4860
'19
MOVJ C01322 BC01322 VJ=100.00  +MOVJ EC01322 VJ=100.00
'Path W4131
SFTOF3D
SFTON3D P023
MOVJ C01323 BC01323 VJ=100.00  +MOVJ EC01323 VJ=100.00
SMOVL C01324 BC01324 V=800.0  +MOVJ EC01324
SMOVL C01325 BC01325 V=166.7 PL=0  +MOVJ EC01325
MACRO1 MJ#(0) ARGF6
ARCON
SWVON WEV#(66)
SMOVL C01326 BC01326 V=7.5  +MOVJ EC01326
SMOVL C01327 BC01327 V=7.5  +MOVJ EC01327
SMOVL C01328 BC01328 V=7.5  +MOVJ EC01328
ARCOF
SWVOF
SMOVL C01329 BC01329 V=800.0  +MOVJ EC01329
SMOVL C01330 BC01330 V=1000.0  +MOVJ EC01330
SFTOF3D
'EndPath W4131
MOVJ C01331 BC01331 VJ=100.00  +MOVJ EC01331 VJ=100.00
'Path W4214
SFTOF3D
SFTON3D P089
MOVJ C01332 BC01332 VJ=100.00  +MOVJ EC01332 VJ=100.00
SMOVL C01333 BC01333 V=800.0  +MOVJ EC01333
SMOVL C01334 BC01334 V=150.0 PL=0  +MOVJ EC01334
MACRO1 MJ#(0) ARGF9
ARCON
SMOVL C01335 BC01335 V=9.2  +MOVJ EC01335
SFTON3D P050
SMOVL C01336 BC01336 V=9.2  +MOVJ EC01336
SMOVL C01337 BC01337 V=9.2  +MOVJ EC01337
ARCOF
SMOVL C01338 BC01338 V=800.0  +MOVJ EC01338
SMOVL C01339 BC01339 V=1000.0  +MOVJ EC01339
SFTOF3D
'EndPath W4214
'Path W4215
SFTOF3D
SFTON3D P051
MOVJ C01340 BC01340 VJ=100.00  +MOVJ EC01340 VJ=100.00
SMOVL C01341 BC01341 V=800.0  +MOVJ EC01341
SMOVL C01342 BC01342 V=150.0 PL=0  +MOVJ EC01342
MACRO1 MJ#(0) ARGF9
ARCON
SWVON WEV#(60)
SMOVL C01343 BC01343 V=7.5  +MOVJ EC01343
SMOVL C01344 BC01344 V=7.5  +MOVJ EC01344
SMOVL C01345 BC01345 V=7.5  +MOVJ EC01345
ARCOF
SWVOF
SMOVL C01346 BC01346 V=800.0  +MOVJ EC01346
SMOVL C01347 BC01347 V=1000.0  +MOVJ EC01347
SFTOF3D
'EndPath W4215
MOVJ C01348 BC01348 VJ=100.00  +MOVJ EC01348 VJ=100.00
'20
'offset 5mm
MOVJ C01349 BC01349 VJ=100.00  +MOVJ EC01349 VJ=100.00
MOVJ C01350 BC01350 VJ=100.00  +MOVJ EC01350 VJ=100.00
'Path W4132
SFTOF3D
SFTON3D P032
MOVJ C01351 BC01351 VJ=100.00  +MOVJ EC01351 VJ=100.00
SMOVL C01352 BC01352 V=800.0  +MOVJ EC01352
SMOVL C01353 BC01353 V=150.0 PL=0  +MOVJ EC01353
ARCON
SMOVL C01354 BC01354 V=10.0  +MOVJ EC01354
SMOVL C01355 BC01355 V=10.0  +MOVJ EC01355
ARCOF
SMOVL C01356 BC01356 V=800.0  +MOVJ EC01356
SMOVL C01357 BC01357 V=1000.0  +MOVJ EC01357
SFTOF3D
JUMP *FFF
'EndPath W4132
'Path W4133
SFTOF3D
SFTON3D P032
MOVJ C01358 BC01358 VJ=100.00  +MOVJ EC01358 VJ=100.00
SMOVL C01359 BC01359 V=800.0  +MOVJ EC01359
SMOVL C01360 BC01360 V=166.7 PL=0  +MOVJ EC01360
ARCON
SMOVL C01361 BC01361 V=10.0  +MOVJ EC01361
ARCOF
SMOVL C01362 BC01362 V=800.0  +MOVJ EC01362
SMOVL C01363 BC01363 V=1000.0  +MOVJ EC01363
SFTOF3D
'EndPath W4133
'Path W4134
SFTOF3D
SFTON3D P032
MOVJ C01364 BC01364 VJ=100.00  +MOVJ EC01364 VJ=100.00
SMOVL C01365 BC01365 V=800.0  +MOVJ EC01365
SMOVL C01366 BC01366 V=150.0 PL=0  +MOVJ EC01366
ARCON
SMOVL C01367 BC01367 V=10.0  +MOVJ EC01367
ARCOF
SMOVL C01368 BC01368 V=800.0  +MOVJ EC01368
*FFF
SMOVL C01369 BC01369 V=1000.0  +MOVJ EC01369
SFTOF3D
'EndPath W4134
'offset 5mm
MOVJ C01370 BC01370 VJ=100.00  +MOVJ EC01370 VJ=100.00
'Path W4135
SFTOF3D
SFTON3D P032
MOVJ C01371 BC01371 VJ=100.00  +MOVJ EC01371 VJ=100.00
SMOVL C01372 BC01372 V=800.0  +MOVJ EC01372
SMOVL C01373 BC01373 V=166.7 PL=0  +MOVJ EC01373
ARCON
SMOVL C01374 BC01374 V=10.0  +MOVJ EC01374
ARCOF
SMOVL C01375 BC01375 V=800.0  +MOVJ EC01375
SMOVL C01376 BC01376 V=1000.0  +MOVJ EC01376
SFTOF3D
'EndPath W4135
MOVJ C01377 BC01377 VJ=100.00  +MOVJ EC01377 VJ=100.00
'Path W4136
SFTOF3D
SFTON3D P032
MOVJ C01378 BC01378 VJ=100.00  +MOVJ EC01378 VJ=100.00
SMOVL C01379 BC01379 V=800.0  +MOVJ EC01379
SMOVL C01380 BC01380 V=166.7 PL=0  +MOVJ EC01380
ARCON
SMOVL C01381 BC01381 V=11.7  +MOVJ EC01381
SMOVL C01382 BC01382 V=11.7  +MOVJ EC01382
ARCOF
SMOVL C01383 BC01383 V=800.0  +MOVJ EC01383
SMOVL C01384 BC01384 V=1000.0  +MOVJ EC01384
SFTOF3D
'EndPath W4136
MOVJ C01385 BC01385 VJ=100.00  +MOVJ EC01385 VJ=100.00
MOVJ C01386 BC01386 VJ=100.00  +MOVJ EC01386 VJ=100.00
'Path W4137
SFTOF3D
SFTON3D P097
MACRO1 MJ#(0) ARGF9
MOVJ C01387 BC01387 VJ=100.00  +MOVJ EC01387 VJ=100.00
SMOVL C01388 BC01388 V=800.0  +MOVJ EC01388
SMOVL C01389 BC01389 V=166.7 PL=0  +MOVJ EC01389
ARCON
SMOVL C01390 BC01390 V=10.0  +MOVJ EC01390
SFTON3D P021
SMOVL C01391 BC01391 V=10.0  +MOVJ EC01391
SFTON3D P022
SMOVL C01392 BC01392 V=10.0  +MOVJ EC01392
SMOVL C01393 BC01393 V=10.0  +MOVJ EC01393
ARCOF
SMOVL C01394 BC01394 V=800.0  +MOVJ EC01394
SMOVL C01395 BC01395 V=1000.0  +MOVJ EC01395
SFTOF3D
'EndPath W4137
MOVJ C01396 BC01396 VJ=100.00  +MOVJ EC01396 VJ=100.00
'Path W4724
SFTOF3D
SFTON3D P095
MOVJ C01397 BC01397 VJ=100.00  +MOVJ EC01397 VJ=100.00
SMOVL C01398 BC01398 V=800.0  +MOVJ EC01398
SMOVL C01399 BC01399 V=150.0 PL=0  +MOVJ EC01399
ARCON
SMOVL C01400 BC01400 V=10.0  +MOVJ EC01400
SMOVL C01401 BC01401 V=10.0  +MOVJ EC01401
SMOVL C01402 BC01402 V=10.0  +MOVJ EC01402
ARCOF
SMOVL C01403 BC01403 V=800.0  +MOVJ EC01403
SMOVL C01404 BC01404 V=1000.0  +MOVJ EC01404
SFTOF3D
'EndPath W4724
'Path W4725
SFTOF3D
SFTON3D P096
MOVJ C01405 BC01405 VJ=100.00  +MOVJ EC01405 VJ=100.00
SMOVL C01406 BC01406 V=800.0  +MOVJ EC01406
SMOVL C01407 BC01407 V=150.0 PL=0  +MOVJ EC01407
ARCON
SMOVL C01408 BC01408 V=10.0  +MOVJ EC01408
SMOVL C01409 BC01409 V=10.0  +MOVJ EC01409
ARCOF
SMOVL C01410 BC01410 V=800.0  +MOVJ EC01410
SMOVL C01411 BC01411 V=1000.0  +MOVJ EC01411
SFTOF3D
'EndPath W4725
MOVJ C01412 BC01412 VJ=100.00  +MOVJ EC01412 VJ=100.00
'Path W4861
SFTOF3D
SFTON3D P071
MOVJ C01413 BC01413 VJ=100.00  +MOVJ EC01413 VJ=100.00
SMOVL C01414 BC01414 V=800.0  +MOVJ EC01414
SMOVL C01415 BC01415 V=150.0 PL=0  +MOVJ EC01415
MACRO1 MJ#(0) ARGF14
ARCON
SMOVL C01416 BC01416 V=9.2  +MOVJ EC01416
SFTON3D P073
SMOVL C01417 BC01417 V=9.2  +MOVJ EC01417
SMOVL C01418 BC01418 V=9.2  +MOVJ EC01418
ARCOF
SMOVL C01419 BC01419 V=800.0  +MOVJ EC01419
SMOVL C01420 BC01420 V=1000.0  +MOVJ EC01420
SFTOF3D
SMOVL C01421 BC01421 V=1000.0  +MOVJ EC01421
SFTOF3D
SFTON3D P080
MOVJ C01422 BC01422 VJ=100.00  +MOVJ EC01422 VJ=100.00
SMOVL C01423 BC01423 V=800.0  +MOVJ EC01423
SMOVL C01424 BC01424 V=150.0 PL=0  +MOVJ EC01424
MACRO1 MJ#(0) ARGF14
ARCON
SMOVL C01425 BC01425 V=9.2  +MOVJ EC01425
SFTON3D P080
SMOVL C01426 BC01426 V=9.2  +MOVJ EC01426
SMOVL C01427 BC01427 V=9.2  +MOVJ EC01427
ARCOF
SMOVL C01428 BC01428 V=800.0  +MOVJ EC01428
SMOVL C01429 BC01429 V=1000.0  +MOVJ EC01429
SFTOF3D
'EndPath W4861
MOVJ C01430 BC01430 VJ=100.00  +MOVJ EC01430 VJ=100.00
MOVJ C01431 BC01431 VJ=100.00  +MOVJ EC01431 VJ=100.00
MOVJ C01432 BC01432 VJ=100.00  +MOVJ EC01432 VJ=100.00
MOVJ C01433 BC01433 VJ=100.00  +MOVJ EC01433 VJ=100.00
MOVJ C01434 BC01434 VJ=100.00  +MOVJ EC01434 VJ=100.00
MOVJ C01435 BC01435 VJ=100.00  +MOVJ EC01435 VJ=100.00
MOVL C01436 BC01436 V=1000.0  +MOVJ EC01436 VJ=100.00
SFTON3D P081
MOVL C01437 BC01437 V=166.7 PL=0  +MOVJ EC01437 VJ=100.00
ARCON
SMOVL C01438 BC01438 V=9.2  +MOVJ EC01438
SMOVL C01439 BC01439 V=9.2  +MOVJ EC01439
SMOVL C01440 BC01440 V=9.2  +MOVJ EC01440
ARCOF
MOVL C01441 BC01441 V=666.7  +MOVJ EC01441 VJ=100.00
SFTOF3D
MOVJ C01442 BC01442 VJ=100.00  +MOVJ EC01442 VJ=100.00
CALL JOB:CLEAN-R1_KM_3P
'cut_wire_dol
'cut_wire_dol
'cut_wire_dol
MOVJ C01443 BC01443 VJ=100.00  +MOVJ EC01443 VJ=100.00
MOVJ C01444 BC01444 VJ=100.00  +MOVJ EC01444 VJ=100.00
MOVJ C01445 BC01445 VJ=100.00  +MOVJ EC01445 VJ=100.00
'Path S4138
SFTOF3D
MOVJ C01446 BC01446 VJ=100.00  +MOVJ EC01446 VJ=100.00
MOVL C01447 BC01447 V=800.0  +MOVJ EC01447 VJ=100.00
SMOVL C01448 BC01448 V=166.7  +MOVJ EC01448
SREFP 3 C01449 BC01449  +REFP EC01449
CALL JOB:SEARCH-R1-S13D
SET P049 P006
SFTON3D P049
SMOVL C01450 BC01450 V=166.7  +MOVJ EC01450
SMOVL C01451 BC01451 V=166.7  +MOVJ EC01451
SREFP 3 C01452 BC01452  +REFP EC01452
CALL JOB:SEARCH-R1-S13D
SET P049 P006
SFTON3D P049
SMOVL C01453 BC01453 V=166.7  +MOVJ EC01453
SMOVL C01454 BC01454 V=166.7  +MOVJ EC01454
SMOVL C01455 BC01455 V=166.7  +MOVJ EC01455
SMOVL C01456 BC01456 V=166.7  +MOVJ EC01456
SREFP 3 C01457 BC01457  +REFP EC01457
CALL JOB:SEARCH-R1-S13D
SET P049 P006
SFTON3D P049
SMOVL C01458 BC01458 V=166.7  +MOVJ EC01458
MOVL C01459 BC01459 V=800.0  +MOVJ EC01459 VJ=100.00
MOVL C01460 BC01460 V=1000.0  +MOVJ EC01460 VJ=100.00
'EndPath S4138
'Path S4139
SFTOF3D
MOVJ C01461 BC01461 VJ=100.00  +MOVJ EC01461 VJ=100.00
MOVL C01462 BC01462 V=800.0  +MOVJ EC01462 VJ=100.00
SMOVL C01463 BC01463 V=166.7  +MOVJ EC01463
SREFP 3 C01464 BC01464  +REFP EC01464
CALL JOB:SEARCH-R1-S13D
SET P048 P006
SFTON3D P048
SMOVL C01465 BC01465 V=166.7  +MOVJ EC01465
SMOVL C01466 BC01466 V=166.7  +MOVJ EC01466
SREFP 3 C01467 BC01467  +REFP EC01467
CALL JOB:SEARCH-R1-S13D
SET P048 P006
SFTON3D P048
SMOVL C01468 BC01468 V=166.7  +MOVJ EC01468
MOVL C01469 BC01469 V=800.0  +MOVJ EC01469 VJ=100.00
MOVL C01470 BC01470 V=1000.0  +MOVJ EC01470 VJ=100.00
'EndPath S4139
'Path S4140
SFTOF3D
MOVJ C01471 BC01471 VJ=100.00  +MOVJ EC01471 VJ=100.00
MOVL C01472 BC01472 V=800.0  +MOVJ EC01472 VJ=100.00
SMOVL C01473 BC01473 V=166.7  +MOVJ EC01473
SREFP 3 C01474 BC01474  +REFP EC01474
CALL JOB:SEARCH-R1-S13D
SET P047 P006
SFTON3D P047
SMOVL C01475 BC01475 V=166.7  +MOVJ EC01475
SMOVL C01476 BC01476 V=166.7  +MOVJ EC01476
SREFP 3 C01477 BC01477  +REFP EC01477
CALL JOB:SEARCH-R1-S13D
SET P047 P006
SFTON3D P047
SMOVL C01478 BC01478 V=166.7  +MOVJ EC01478
MOVL C01479 BC01479 V=800.0  +MOVJ EC01479 VJ=100.00
MOVL C01480 BC01480 V=1000.0  +MOVJ EC01480 VJ=100.00
'EndPath S4140
MOVJ C01481 BC01481 VJ=100.00  +MOVJ EC01481 VJ=100.00
MOVJ C01482 BC01482 VJ=100.00  +MOVJ EC01482 VJ=100.00
MOVJ C01483 BC01483 VJ=100.00  +MOVJ EC01483 VJ=100.00
MOVJ C01484 BC01484 VJ=100.00  +MOVJ EC01484 VJ=100.00
'Path S4141
SFTOF3D
MOVJ C01485 BC01485 VJ=100.00  +MOVJ EC01485 VJ=100.00
MOVL C01486 BC01486 V=800.0  +MOVJ EC01486 VJ=100.00
SMOVL C01487 BC01487 V=166.7  +MOVJ EC01487
SREFP 3 C01488 BC01488  +REFP EC01488
CALL JOB:SEARCH-R1-S13D
SET P046 P006
SFTON3D P046
SMOVL C01489 BC01489 V=166.7  +MOVJ EC01489
SMOVL C01490 BC01490 V=166.7  +MOVJ EC01490
SREFP 3 C01491 BC01491  +REFP EC01491
CALL JOB:SEARCH-R1-S13D
SET P046 P006
SFTON3D P046
SMOVL C01492 BC01492 V=166.7  +MOVJ EC01492
MOVL C01493 BC01493 V=1000.0  +MOVJ EC01493 VJ=100.00
'EndPath S4141
'Path S4142
SFTOF3D
MOVJ C01494 BC01494 VJ=100.00  +MOVJ EC01494 VJ=100.00
MOVL C01495 BC01495 V=800.0  +MOVJ EC01495 VJ=100.00
SMOVL C01496 BC01496 V=166.7  +MOVJ EC01496
SREFP 3 C01497 BC01497  +REFP EC01497
CALL JOB:SEARCH-R1-S13D
SET P055 P006
SFTON3D P055
SMOVL C01498 BC01498 V=166.7  +MOVJ EC01498
SMOVL C01499 BC01499 V=166.7  +MOVJ EC01499
SMOVL C01500 BC01500 V=166.7  +MOVJ EC01500
SREFP 3 C01501 BC01501  +REFP EC01501
CALL JOB:SEARCH-R1-S13D
SET P055 P006
SFTON3D P055
SMOVL C01502 BC01502 V=166.7  +MOVJ EC01502
SREFP 3 C01503 BC01503  +REFP EC01503
CALL JOB:SEARCH-R1-S13D
SET P045 P006
SFTON3D P045
SMOVL C01504 BC01504 V=166.7  +MOVJ EC01504
SMOVL C01505 BC01505 V=166.7  +MOVJ EC01505
SMOVL C01506 BC01506 V=166.7  +MOVJ EC01506
SREFP 3 C01507 BC01507  +REFP EC01507
CALL JOB:SEARCH-R1-S13D
SET P045 P006
SFTON3D P045
SMOVL C01508 BC01508 V=166.7  +MOVJ EC01508
MOVL C01509 BC01509 V=1000.0  +MOVJ EC01509 VJ=100.00
'EndPath S4142
'Path S4143
SFTOF3D
MOVJ C01510 BC01510 VJ=100.00  +MOVJ EC01510 VJ=100.00
MOVL C01511 BC01511 V=800.0  +MOVJ EC01511 VJ=100.00
SMOVL C01512 BC01512 V=166.7  +MOVJ EC01512
SREFP 3 C01513 BC01513  +REFP EC01513
CALL JOB:SEARCH-R1-S13D
SET P054 P006
SFTON3D P054
SMOVL C01514 BC01514 V=166.7  +MOVJ EC01514
SMOVL C01515 BC01515 V=166.7  +MOVJ EC01515
SMOVL C01516 BC01516 V=166.7  +MOVJ EC01516
SREFP 3 C01517 BC01517  +REFP EC01517
CALL JOB:SEARCH-R1-S13D
SET P054 P006
SFTON3D P054
SMOVL C01518 BC01518 V=166.7  +MOVJ EC01518
SREFP 3 C01519 BC01519  +REFP EC01519
CALL JOB:SEARCH-R1-S13D
SET P044 P006
SFTON3D P044
SMOVL C01520 BC01520 V=166.7  +MOVJ EC01520
SMOVL C01521 BC01521 V=166.7  +MOVJ EC01521
MOVL C01522 BC01522 V=166.7  +MOVJ EC01522 VJ=0.78
SREFP 3 C01523 BC01523  +REFP EC01523
CALL JOB:SEARCH-R1-S13D
SET P044 P006
SFTON3D P044
SMOVL C01524 BC01524 V=166.7  +MOVJ EC01524
MOVL C01525 BC01525 V=1000.0  +MOVJ EC01525 VJ=100.00
'EndPath S4143
MOVJ C01526 BC01526 VJ=100.00  +MOVJ EC01526 VJ=100.00
MOVJ C01527 BC01527 VJ=100.00  +MOVJ EC01527 VJ=100.00
'Path S4144
SFTOF3D
MOVJ C01528 BC01528 VJ=100.00  +MOVJ EC01528 VJ=100.00
MOVL C01529 BC01529 V=800.0  +MOVJ EC01529 VJ=100.00
SMOVL C01530 BC01530 V=166.7  +MOVJ EC01530
SREFP 3 C01531 BC01531  +REFP EC01531
CALL JOB:SEARCH-R1-S13D
SET P053 P006
SFTON3D P053
SMOVL C01532 BC01532 V=166.7  +MOVJ EC01532
SMOVL C01533 BC01533 V=166.7  +MOVJ EC01533
MOVL C01534 BC01534 V=166.7  +MOVJ EC01534 VJ=0.78
SREFP 3 C01535 BC01535  +REFP EC01535
CALL JOB:SEARCH-R1-S13D
SET P053 P006
SFTON3D P053
SMOVL C01536 BC01536 V=166.7  +MOVJ EC01536
SREFP 3 C01537 BC01537  +REFP EC01537
CALL JOB:SEARCH-R1-S13D
SET P043 P006
SFTON3D P043
SMOVL C01538 BC01538 V=166.7  +MOVJ EC01538
SMOVL C01539 BC01539 V=166.7  +MOVJ EC01539
MOVL C01540 BC01540 V=166.7  +MOVJ EC01540 VJ=0.78
SREFP 3 C01541 BC01541  +REFP EC01541
CALL JOB:SEARCH-R1-S13D
SET P043 P006
SFTON3D P043
SMOVL C01542 BC01542 V=166.7  +MOVJ EC01542
MOVL C01543 BC01543 V=1000.0  +MOVJ EC01543 VJ=100.00
'EndPath S4144
'Path S4145
SFTOF3D
MOVJ C01544 BC01544 VJ=100.00  +MOVJ EC01544 VJ=100.00
MOVL C01545 BC01545 V=800.0  +MOVJ EC01545 VJ=100.00
SMOVL C01546 BC01546 V=166.7  +MOVJ EC01546
SREFP 3 C01547 BC01547  +REFP EC01547
CALL JOB:SEARCH-R1-S13D
SET P052 P006
SFTON3D P052
SMOVL C01548 BC01548 V=166.7  +MOVJ EC01548
SMOVL C01549 BC01549 V=166.7  +MOVJ EC01549
MOVL C01550 BC01550 V=166.7  +MOVJ EC01550 VJ=0.78
SREFP 3 C01551 BC01551  +REFP EC01551
CALL JOB:SEARCH-R1-S13D
SET P052 P006
SFTON3D P052
SMOVL C01552 BC01552 V=166.7  +MOVJ EC01552
SREFP 3 C01553 BC01553  +REFP EC01553
CALL JOB:SEARCH-R1-S13D
SET P042 P006
SFTON3D P042
SMOVL C01554 BC01554 V=166.7  +MOVJ EC01554
SMOVL C01555 BC01555 V=166.7  +MOVJ EC01555
MOVL C01556 BC01556 V=166.7  +MOVJ EC01556 VJ=0.78
SREFP 3 C01557 BC01557  +REFP EC01557
CALL JOB:SEARCH-R1-S13D
SET P042 P006
SFTON3D P042
SMOVL C01558 BC01558 V=166.7  +MOVJ EC01558
MOVL C01559 BC01559 V=1000.0  +MOVJ EC01559 VJ=100.00
'EndPath S4145
'Path S4146
SFTOF3D
MOVJ C01560 BC01560 VJ=100.00  +MOVJ EC01560 VJ=100.00
MOVL C01561 BC01561 V=666.7  +MOVJ EC01561 VJ=100.00
SMOVL C01562 BC01562 V=166.7  +MOVJ EC01562
SREFP 3 C01563 BC01563  +REFP EC01563
CALL JOB:SEARCH-R1-S13D
SET P041 P006
SFTON3D P041
SMOVL C01564 BC01564 V=250.0  +MOVJ EC01564
SMOVL C01565 BC01565 V=166.7  +MOVJ EC01565
SREFP 3 C01566 BC01566  +REFP EC01566
CALL JOB:SEARCH-R1-S13D
SET P041 P006
SFTON3D P041
SMOVL C01567 BC01567 V=166.7  +MOVJ EC01567
SMOVL C01568 BC01568 V=166.7  +MOVJ EC01568
SREFP 3 C01569 BC01569  +REFP EC01569
CALL JOB:SEARCH-R1-S13D
SET P041 P006
SFTON3D P041
SMOVL C01570 BC01570 V=166.7  +MOVJ EC01570
MOVL C01571 BC01571 V=1000.0  +MOVJ EC01571 VJ=100.00
'EndPath S4146
'Path S4147
SFTOF3D
MOVJ C01572 BC01572 VJ=100.00  +MOVJ EC01572 VJ=100.00
SMOVL C01573 BC01573 V=666.7  +MOVJ EC01573
SMOVL C01574 BC01574 V=166.7  +MOVJ EC01574
SREFP 3 C01575 BC01575  +REFP EC01575
CALL JOB:SEARCH-R1-S13D
SET P040 P006
SFTON3D P040
SMOVL C01576 BC01576 V=166.7  +MOVJ EC01576
SMOVL C01577 BC01577 V=800.0  +MOVJ EC01577
SMOVL C01578 BC01578 V=166.7  +MOVJ EC01578
SREFP 3 C01579 BC01579  +REFP EC01579
CALL JOB:SEARCH-R1-S13D
SET P040 P006
SFTON3D P040
SMOVL C01580 BC01580 V=166.7  +MOVJ EC01580
SMOVL C01581 BC01581 V=166.7  +MOVJ EC01581
SREFP 3 C01582 BC01582  +REFP EC01582
CALL JOB:SEARCH-R1-S13D
SET P040 P006
SFTON3D P040
SMOVL C01583 BC01583 V=166.7  +MOVJ EC01583
MOVL C01584 BC01584 V=1000.0  +MOVJ EC01584 VJ=100.00
'EndPath S4147
'Path W4148
SFTOF3D
SFTON3D P040
MOVJ C01585 BC01585 VJ=100.00  +MOVJ EC01585 VJ=100.00
SMOVL C01586 BC01586 V=800.0  +MOVJ EC01586
SMOVL C01587 BC01587 V=150.0 PL=0  +MOVJ EC01587
ARCON
SMOVL C01588 BC01588 V=10.0  +MOVJ EC01588
ARCOF
SMOVL C01589 BC01589 V=800.0  +MOVJ EC01589
SMOVL C01590 BC01590 V=1000.0  +MOVJ EC01590
SFTOF3D
'EndPath W4148
'Path W4149
SFTOF3D
SFTON3D P040
MOVJ C01591 BC01591 VJ=100.00  +MOVJ EC01591 VJ=100.00
SMOVL C01592 BC01592 V=800.0  +MOVJ EC01592
SMOVL C01593 BC01593 V=150.0 PL=0  +MOVJ EC01593
ARCON
SMOVL C01594 BC01594 V=11.7  +MOVJ EC01594
ARCOF
SMOVL C01595 BC01595 V=800.0  +MOVJ EC01595
SMOVL C01596 BC01596 V=1000.0  +MOVJ EC01596
SFTOF3D
'EndPath W4149
'Path W4150
SFTOF3D
SFTON3D P040
MOVJ C01597 BC01597 VJ=15.00  +MOVJ EC01597 VJ=15.00
MOVJ C01598 BC01598 VJ=100.00  +MOVJ EC01598 VJ=100.00
SMOVL C01599 BC01599 V=800.0  +MOVJ EC01599
SMOVL C01600 BC01600 V=150.0 PL=0  +MOVJ EC01600
ARCON
SMOVL C01601 BC01601 V=11.7  +MOVJ EC01601
ARCOF
SMOVL C01602 BC01602 V=800.0  +MOVJ EC01602
SMOVL C01603 BC01603 V=1000.0  +MOVJ EC01603
SFTOF3D
'EndPath W4150
'
MOVJ C01604 BC01604 VJ=100.00  +MOVJ EC01604 VJ=100.00
MOVJ C01605 BC01605 VJ=100.00  +MOVJ EC01605 VJ=100.00
'Path W4151
SFTOF3D
SFTON3D P045
MOVJ C01606 BC01606 VJ=100.00  +MOVJ EC01606 VJ=100.00
SMOVL C01607 BC01607 V=800.0  +MOVJ EC01607
SMOVL C01608 BC01608 V=150.0 PL=0  +MOVJ EC01608
MACRO1 MJ#(0) ARGF9
ARCON
SMOVL C01609 BC01609 V=11.7  +MOVJ EC01609
ARCOF
SMOVL C01610 BC01610 V=800.0  +MOVJ EC01610
SMOVL C01611 BC01611 V=1000.0  +MOVJ EC01611
SFTOF3D
'EndPath W4151
'Path W4152
SFTOF3D
SFTON3D P044
MOVJ C01612 BC01612 VJ=100.00  +MOVJ EC01612 VJ=100.00
SMOVL C01613 BC01613 V=800.0  +MOVJ EC01613
SMOVL C01614 BC01614 V=166.7 PL=0  +MOVJ EC01614
ARCON
SMOVL C01615 BC01615 V=11.7  +MOVJ EC01615
ARCOF
SMOVL C01616 BC01616 V=800.0  +MOVJ EC01616
SMOVL C01617 BC01617 V=1000.0  +MOVJ EC01617
SFTOF3D
'EndPath W4152
'Path W4153
SFTOF3D
SFTON3D P046
MOVJ C01618 BC01618 VJ=100.00  +MOVJ EC01618 VJ=100.00
SMOVL C01619 BC01619 V=800.0  +MOVJ EC01619
SMOVL C01620 BC01620 V=166.7 PL=0  +MOVJ EC01620
MACRO1 MJ#(0) ARGF14
ARCON
SMOVL C01621 BC01621 V=10.0  +MOVJ EC01621
SMOVL C01622 BC01622 V=10.0  +MOVJ EC01622
ARCOF
SMOVL C01623 BC01623 V=800.0  +MOVJ EC01623
SMOVL C01624 BC01624 V=1000.0  +MOVJ EC01624
SFTOF3D
'EndPath W4153
MOVJ C01625 BC01625 VJ=100.00  +MOVJ EC01625 VJ=100.00
MOVJ C01626 BC01626 VJ=100.00  +MOVJ EC01626 VJ=100.00
MOVJ C01627 BC01627 VJ=100.00  +MOVJ EC01627 VJ=100.00
MOVJ C01628 BC01628 VJ=100.00  +MOVJ EC01628 VJ=100.00
'1
'uwaga na podajnik
'Path W4154
SFTOF3D
SFTON3D P048
MOVJ C01629 BC01629 VJ=100.00  +MOVJ EC01629 VJ=100.00
SMOVL C01630 BC01630 V=800.0  +MOVJ EC01630
SMOVL C01631 BC01631 V=150.0 PL=0  +MOVJ EC01631
ARCON
SMOVL C01632 BC01632 V=10.0  +MOVJ EC01632
ARCOF
SMOVL C01633 BC01633 V=800.0  +MOVJ EC01633
SMOVL C01634 BC01634 V=1000.0  +MOVJ EC01634
SFTOF3D
'EndPath W4154
'Path W4155
SFTOF3D
SFTON3D P049
MOVJ C01635 BC01635 VJ=100.00  +MOVJ EC01635 VJ=100.00
SMOVL C01636 BC01636 V=800.0  +MOVJ EC01636
SMOVL C01637 BC01637 V=150.0 PL=0  +MOVJ EC01637
MACRO1 MJ#(0) ARGF6
ARCON
SMOVL C01638 BC01638 V=9.2  +MOVJ EC01638
SMOVL C01639 BC01639 V=9.2  +MOVJ EC01639
SMOVL C01640 BC01640 V=9.2  +MOVJ EC01640
SMOVL C01641 BC01641 V=9.2  +MOVJ EC01641
SMOVL C01642 BC01642 V=9.2  +MOVJ EC01642
ARCOF
SMOVL C01643 BC01643 V=800.0  +MOVJ EC01643
SMOVL C01644 BC01644 V=500.0  +MOVJ EC01644
SMOVL C01645 BC01645 V=133.3  +MOVJ EC01645
ARCON
SMOVL C01646 BC01646 V=13.3  +MOVJ EC01646
ARCOF
SMOVL C01647 BC01647 V=166.7  +MOVJ EC01647
ARCON
SMOVL C01648 BC01648 V=10.0  +MOVJ EC01648
ARCOF
SMOVL C01649 BC01649 V=250.0  +MOVJ EC01649
SMOVL C01650 BC01650 V=500.0  +MOVJ EC01650
SMOVL C01651 BC01651 V=500.0  +MOVJ EC01651
SMOVL C01652 BC01652 V=500.0  +MOVJ EC01652
SMOVL C01653 BC01653 V=133.3  +MOVJ EC01653
ARCON
SMOVL C01654 BC01654 V=13.3  +MOVJ EC01654
ARCOF
SMOVL C01655 BC01655 V=166.7  +MOVJ EC01655
SMOVL C01656 BC01656 V=166.7  +MOVJ EC01656
ARCON
SMOVL C01657 BC01657 V=10.0  +MOVJ EC01657
ARCOF
SMOVL C01658 BC01658 V=800.0  +MOVJ EC01658
SFTOF3D
'EndPath W4155
MOVJ C01659 BC01659 VJ=100.00  +MOVJ EC01659 VJ=100.00
MOVJ C01660 BC01660 VJ=100.00  +MOVJ EC01660 VJ=100.00
MOVJ C01661 BC01661 VJ=100.00  +MOVJ EC01661 VJ=100.00
MOVJ C01662 BC01662 VJ=100.00  +MOVJ EC01662 VJ=100.00
'2
'Path W4156
SFTOF3D
SFTON3D P043
MOVJ C01663 BC01663 VJ=100.00  +MOVJ EC01663 VJ=100.00
SMOVL C01664 BC01664 V=800.0  +MOVJ EC01664
SMOVL C01665 BC01665 V=166.7 PL=0  +MOVJ EC01665
MACRO1 MJ#(0) ARGF9
ARCON
SMOVL C01666 BC01666 V=11.7  +MOVJ EC01666
ARCOF
SMOVL C01667 BC01667 V=800.0  +MOVJ EC01667
SMOVL C01668 BC01668 V=1000.0  +MOVJ EC01668
SFTOF3D
'EndPath W4156
'Path W4157
SFTOF3D
SFTON3D P042
MOVJ C01669 BC01669 VJ=100.00  +MOVJ EC01669 VJ=100.00
SMOVL C01670 BC01670 V=800.0  +MOVJ EC01670
SMOVL C01671 BC01671 V=150.0 PL=0  +MOVJ EC01671
ARCON
SMOVL C01672 BC01672 V=11.7  +MOVJ EC01672
ARCOF
SMOVL C01673 BC01673 V=800.0  +MOVJ EC01673
SMOVL C01674 BC01674 V=1000.0  +MOVJ EC01674
SFTOF3D
'EndPath W4157
'3
MOVJ C01675 BC01675 VJ=100.00  +MOVJ EC01675 VJ=100.00
MOVJ C01676 BC01676 VJ=100.00  +MOVJ EC01676 VJ=100.00
MOVJ C01677 BC01677 VJ=100.00  +MOVJ EC01677 VJ=100.00
MOVJ C01678 BC01678 VJ=100.00  +MOVJ EC01678 VJ=100.00
'Path W4158
SFTOF3D
SFTON3D P047
MOVJ C01679 BC01679 VJ=100.00  +MOVJ EC01679 VJ=100.00
SMOVL C01680 BC01680 V=800.0  +MOVJ EC01680
SMOVL C01681 BC01681 V=150.0 PL=0  +MOVJ EC01681
ARCON
SMOVL C01682 BC01682 V=11.7  +MOVJ EC01682
ARCOF
SMOVL C01683 BC01683 V=800.0  +MOVJ EC01683
SMOVL C01684 BC01684 V=1000.0  +MOVJ EC01684
SFTOF3D
'EndPath W4158
'Path W4159
SFTOF3D
SFTON3D P047
MOVJ C01685 BC01685 VJ=100.00  +MOVJ EC01685 VJ=100.00
SMOVL C01686 BC01686 V=800.0  +MOVJ EC01686
SMOVL C01687 BC01687 V=150.0 PL=0  +MOVJ EC01687
ARCON
SMOVL C01688 BC01688 V=11.7  +MOVJ EC01688
ARCOF
SMOVL C01689 BC01689 V=800.0  +MOVJ EC01689
SMOVL C01690 BC01690 V=1000.0  +MOVJ EC01690
SFTOF3D
'EndPath W4159
MOVJ C01691 BC01691 VJ=100.00  +MOVJ EC01691 VJ=100.00
MOVJ C01692 BC01692 VJ=100.00  +MOVJ EC01692 VJ=100.00
MOVJ C01693 BC01693 VJ=100.00  +MOVJ EC01693 VJ=100.00
MOVJ C01694 BC01694 VJ=100.00  +MOVJ EC01694 VJ=100.00
'Path W4160
SFTOF3D
SFTON3D P043
MOVJ C01695 BC01695 VJ=100.00  +MOVJ EC01695 VJ=100.00
SMOVL C01696 BC01696 V=800.0  +MOVJ EC01696
SMOVL C01697 BC01697 V=150.0 PL=0  +MOVJ EC01697
ARCON
SMOVL C01698 BC01698 V=11.7  +MOVJ EC01698
ARCOF
SMOVL C01699 BC01699 V=800.0  +MOVJ EC01699
SMOVL C01700 BC01700 V=1000.0  +MOVJ EC01700
SFTOF3D
'EndPath W4160
'Path W4161
SFTOF3D
SFTON3D P042
MOVJ C01701 BC01701 VJ=100.00  +MOVJ EC01701 VJ=100.00
SMOVL C01702 BC01702 V=800.0  +MOVJ EC01702
SMOVL C01703 BC01703 V=166.7 PL=0  +MOVJ EC01703
ARCON
SMOVL C01704 BC01704 V=11.7  +MOVJ EC01704
ARCOF
SMOVL C01705 BC01705 V=800.0  +MOVJ EC01705
SMOVL C01706 BC01706 V=1000.0  +MOVJ EC01706
SFTOF3D
'EndPath W4161
MOVJ C01707 BC01707 VJ=100.00  +MOVJ EC01707 VJ=100.00
'Path W4162
SFTOF3D
SFTON3D P046
MOVJ C01708 BC01708 VJ=100.00  +MOVJ EC01708 VJ=100.00
SMOVL C01709 BC01709 V=800.0  +MOVJ EC01709
SMOVL C01710 BC01710 V=166.7 PL=0  +MOVJ EC01710
MACRO1 MJ#(0) ARGF14
ARCON
SMOVL C01711 BC01711 V=10.0  +MOVJ EC01711
ARCOF
SMOVL C01712 BC01712 V=800.0  +MOVJ EC01712
SMOVL C01713 BC01713 V=1000.0  +MOVJ EC01713
SFTOF3D
'EndPath W4162
'Path W4163
SFTOF3D
SFTON3D P044
MOVJ C01714 BC01714 VJ=100.00  +MOVJ EC01714 VJ=100.00
SMOVL C01715 BC01715 V=800.0  +MOVJ EC01715
SMOVL C01716 BC01716 V=150.0 PL=0  +MOVJ EC01716
MACRO1 MJ#(0) ARGF9
ARCON
SMOVL C01717 BC01717 V=11.7  +MOVJ EC01717
ARCOF
SMOVL C01718 BC01718 V=800.0  +MOVJ EC01718
SMOVL C01719 BC01719 V=1000.0  +MOVJ EC01719
SFTOF3D
'EndPath W4163
MOVJ C01720 BC01720 VJ=100.00  +MOVJ EC01720 VJ=100.00
'Path W4164
SFTOF3D
SFTON3D P041
MOVJ C01721 BC01721 VJ=100.00  +MOVJ EC01721 VJ=100.00
SMOVL C01722 BC01722 V=800.0  +MOVJ EC01722
SMOVL C01723 BC01723 V=150.0 PL=0  +MOVJ EC01723
MACRO1 MJ#(0) ARGF14
ARCON
SMOVL C01724 BC01724 V=10.0  +MOVJ EC01724
SMOVL C01725 BC01725 V=10.0  +MOVJ EC01725
SMOVL C01726 BC01726 V=10.0  +MOVJ EC01726
ARCOF
SMOVL C01727 BC01727 V=800.0  +MOVJ EC01727
SMOVL C01728 BC01728 V=1000.0  +MOVJ EC01728
SFTOF3D
'EndPath W4164
JUMP *L_1
'Path W4165
SFTOF3D
SFTON3D P041
MOVJ C01729 BC01729 VJ=100.00  +MOVJ EC01729 VJ=100.00
SMOVL C01730 BC01730 V=800.0  +MOVJ EC01730
SMOVL C01731 BC01731 V=150.0 PL=0  +MOVJ EC01731
SMOVL C01732 BC01732 V=10.0  +MOVJ EC01732
ARCOF
SMOVL C01733 BC01733 V=800.0  +MOVJ EC01733
SMOVL C01734 BC01734 V=1000.0  +MOVJ EC01734
SFTOF3D
'EndPath W4165
MOVJ C01735 BC01735 VJ=100.00  +MOVJ EC01735 VJ=100.00
'Path W4166
SFTOF3D
SFTON3D P041
MOVJ C01736 BC01736 VJ=100.00  +MOVJ EC01736 VJ=100.00
SMOVL C01737 BC01737 V=800.0  +MOVJ EC01737
SMOVL C01738 BC01738 V=150.0 PL=0  +MOVJ EC01738
SMOVL C01739 BC01739 V=10.0  +MOVJ EC01739
ARCOF
SMOVL C01740 BC01740 V=800.0  +MOVJ EC01740
SMOVL C01741 BC01741 V=1000.0  +MOVJ EC01741
SFTOF3D
'EndPath W4166
*L_1
MOVJ C01742 BC01742 VJ=100.00  +MOVJ EC01742 VJ=100.00
MOVJ C01743 BC01743 VJ=100.00  +MOVJ EC01743 VJ=100.00
MOVJ C01744 BC01744 VJ=100.00  +MOVJ EC01744 VJ=100.00
END
